LIN {X 0,Y 486.254,Z 781.859,A -85,B 0,C 180,E1 22613.17,E2 22613.17} C_VEL
LIN {X 0,Y 485.416,Z 799.484,A -85,B 0,C 180,E1 22612.272,E2 22612.272} C_VEL
LIN {X 0,Y 484.471,Z 816.535,A -85,B 0,C 180,E1 22611.172,E2 22611.172} C_VEL
LIN {X 0,Y 483.537,Z 833.395,A -85,B 0,C 180,E1 22609.824,E2 22609.824} C_VEL
LIN {X 0,Y 482.628,Z 848.999,A -85,B 0,C 180,E1 22608.302,E2 22608.302} C_VEL
LIN {X 0,Y 481.853,Z 863.116,A -85,B 0,C 180,E1 22606.64,E2 22606.64} C_VEL
LIN {X 0,Y 481.192,Z 876.044,A -85,B 0,C 180,E1 22604.808,E2 22604.808} C_VEL
LIN {X 0,Y 480.699,Z 887.391,A -85,B 0,C 180,E1 22602.86,E2 22602.86} C_VEL
LIN {X 0,Y 480.358,Z 897.146,A -85,B 0,C 180,E1 22600.797,E2 22600.797} C_VEL
LIN {X 0,Y 480.152,Z 905.245,A -85,B 0,C 180,E1 22598.623,E2 22598.623} C_VEL
LIN {X 0,Y 480.072,Z 911.354,A -85,B 0,C 180,E1 22596.458,E2 22596.458} C_VEL
LIN {X 0,Y 480.048,Z 915.622,A -85,B 0,C 180,E1 22594.3,E2 22594.3} C_VEL
LIN {X 0,Y 480.043,Z 918.148,A -85,B 0,C 180,E1 22592.149,E2 22592.149} C_VEL
LIN {X 0,Y 480.045,Z 918.986,A -85,B 0,C 180,E1 22590,E2 22590} C_VEL
LIN {X 0,Y 480.041,Z 918.046,A -85,B 0,C 180,E1 22587.732,E2 22587.732} C_VEL
LIN {X 0,Y 480.048,Z 915.422,A -85,B 0,C 180,E1 22585.58,E2 22585.58} C_VEL
LIN {X 0,Y 480.074,Z 911.042,A -85,B 0,C 180,E1 22583.423,E2 22583.423} C_VEL
LIN {X 0,Y 480.159,Z 904.804,A -85,B 0,C 180,E1 22581.257,E2 22581.257} C_VEL
LIN {X 0,Y 480.363,Z 897.052,A -85,B 0,C 180,E1 22579.203,E2 22579.203} C_VEL
LIN {X 0,Y 480.7,Z 887.258,A -85,B 0,C 180,E1 22577.141,E2 22577.141} C_VEL
LIN {X 0,Y 481.191,Z 875.865,A -85,B 0,C 180,E1 22575.192,E2 22575.192} C_VEL
LIN {X 0,Y 481.823,Z 863.363,A -85,B 0,C 180,E1 22573.421,E2 22573.421} C_VEL
LIN {X 0,Y 482.577,Z 849.357,A -85,B 0,C 180,E1 22571.769,E2 22571.769} C_VEL
LIN {X 0,Y 483.439,Z 834.399,A -85,B 0,C 180,E1 22570.299,E2 22570.299} C_VEL
LIN {X 0,Y 484.304,Z 818.578,A -85,B 0,C 180,E1 22569.011,E2 22569.011} C_VEL
LIN {X 0,Y 485.221,Z 801.998,A -85,B 0,C 180,E1 22567.91,E2 22567.91} C_VEL
LIN {X 0,Y 486.072,Z 783.949,A -85,B 0,C 180,E1 22566.959,E2 22566.959} C_VEL
LIN {X 0,Y 486.851,Z 764.903,A -85,B 0,C 180,E1 22566.207,E2 22566.207} C_VEL
LIN {X 0,Y 487.467,Z 746.066,A -85,B 0,C 180,E1 22565.697,E2 22565.697} C_VEL
LIN {X 0,Y 487.855,Z 712.64,A -85,B 0,C 180,E1 22565.166,E2 22565.166} C_VEL
LIN {X 0,Y 489.112,Z 554.122,A -85,B 0,C 180,E1 22562.794,E2 22562.794} C_VEL
LIN {X 0,Y 487.309,Z 539.68,A -85,B 0,C 180,E1 22562.457,E2 22562.457} C_VEL
LIN {X 0,Y 489.579,Z 496.19,A -85,B 0,C 180,E1 22558.839,E2 22558.839} C_VEL
LIN {X 0,Y 490.971,Z 471.845,A -85,B 0,C 180,E1 22556.729,E2 22556.729} C_VEL
LIN {X 0,Y 484.233,Z 452.154,A -85,B 0,C 180,E1 22554.342,E2 22554.342} C_VEL
LIN {X 0,Y 480.918,Z 443.105,A -85,B 0,C 180,E1 22553.11,E2 22553.11} C_VEL
LIN {X 0,Y 480.88,Z 442.893,A -85,B 0,C 180,E1 22549.552,E2 22549.552} C_VEL
LIN {X 0,Y 480.889,Z 442.899,A -85,B 0,C 180,E1 22546.005,E2 22546.005} C_VEL
LIN {X 0,Y 480.884,Z 442.893,A -85,B 0,C 180,E1 22542.35,E2 22542.35} C_VEL
LIN {X 0,Y 480.891,Z 442.887,A -85,B 0,C 180,E1 22538.743,E2 22538.743} C_VEL
LIN {X 0,Y 480.877,Z 442.894,A -85,B 0,C 180,E1 22535.166,E2 22535.166} C_VEL
LIN {X 0,Y 480.881,Z 442.893,A -85,B 0,C 180,E1 22531.518,E2 22531.518} C_VEL
LIN {X 0,Y 480.889,Z 442.887,A -85,B 0,C 180,E1 22527.893,E2 22527.893} C_VEL
LIN {X 0,Y 480.886,Z 442.888,A -85,B 0,C 180,E1 22524.31,E2 22524.31} C_VEL
LIN {X 0,Y 480.883,Z 442.891,A -85,B 0,C 180,E1 22520.699,E2 22520.699} C_VEL
LIN {X 0,Y 480.876,Z 442.897,A -85,B 0,C 180,E1 22517.048,E2 22517.048} C_VEL
LIN {X 0,Y 480.889,Z 442.888,A -85,B 0,C 180,E1 22513.466,E2 22513.466} C_VEL
LIN {X 0,Y 480.884,Z 442.886,A -85,B 0,C 180,E1 22509.816,E2 22509.816} C_VEL
LIN {X 0,Y 480.888,Z 442.891,A -85,B 0,C 180,E1 22506.207,E2 22506.207} C_VEL
LIN {X 0,Y 480.873,Z 442.896,A -85,B 0,C 180,E1 22502.622,E2 22502.622} C_VEL
LIN {X 0,Y 480.887,Z 442.888,A -85,B 0,C 180,E1 22499.047,E2 22499.047} C_VEL
LIN {X 0,Y 480.885,Z 442.889,A -85,B 0,C 180,E1 22495.468,E2 22495.468} C_VEL
LIN {X 0,Y 480.889,Z 442.892,A -85,B 0,C 180,E1 22491.872,E2 22491.872} C_VEL
LIN {X 0,Y 480.872,Z 442.896,A -85,B 0,C 180,E1 22488.242,E2 22488.242} C_VEL
LIN {X 0,Y 480.879,Z 442.899,A -85,B 0,C 180,E1 22484.565,E2 22484.565} C_VEL
LIN {X 0,Y 480.888,Z 442.895,A -85,B 0,C 180,E1 22480.947,E2 22480.947} C_VEL
LIN {X 0,Y 480.893,Z 442.894,A -85,B 0,C 180,E1 22477.378,E2 22477.378} C_VEL
LIN {X 0,Y 480.873,Z 442.897,A -85,B 0,C 180,E1 22473.845,E2 22473.845} C_VEL
LIN {X 0,Y 480.876,Z 442.894,A -85,B 0,C 180,E1 22470.202,E2 22470.202} C_VEL
LIN {X 0,Y 480.892,Z 442.899,A -85,B 0,C 180,E1 22466.565,E2 22466.565} C_VEL
LIN {X 0,Y 480.89,Z 442.9,A -85,B 0,C 180,E1 22462.917,E2 22462.917} C_VEL
LIN {X 0,Y 480.983,Z 443.47,A -85,B 0,C 180,E1 22462.626,E2 22462.626} C_VEL
LIN {X 0,Y 485.678,Z 459.122,A -85,B 0,C 180,E1 22459.981,E2 22459.981} C_VEL
LIN {X 0,Y 487.767,Z 467.746,A -85,B 0,C 180,E1 22458.612,E2 22458.612} C_VEL
LIN {X 0,Y 485.992,Z 496.046,A -85,B 0,C 180,E1 22454.884,E2 22454.884} C_VEL
LIN {X 0,Y 484.498,Z 525.084,A -85,B 0,C 180,E1 22451.127,E2 22451.127} C_VEL
LIN {X 0,Y 483.217,Z 552.995,A -85,B 0,C 180,E1 22447.58,E2 22447.58} C_VEL
LIN {X 0,Y 483.229,Z 556.14,A -85,B 0,C 180,E1 22447.246,E2 22447.246} C_VEL
LIN {X 0,Y 484.694,Z 563.985,A -85,B 0,C 180,E1 22447.03,E2 22447.03} C_VEL
LIN {X 0,Y 484.537,Z 568.371,A -85,B 0,C 180,E1 22446.968,E2 22446.968} C_VEL
LIN {X 0,Y 481.971,Z 575.469,A -85,B 0,C 180,E1 22446.983,E2 22446.983} C_VEL
LIN {X 0,Y 478.786,Z 583.343,A -85,B 0,C 180,E1 22447.017,E2 22447.017} C_VEL
LIN {X 0,Y 478.245,Z 587.099,A -85,B 0,C 180,E1 22446.983,E2 22446.983} C_VEL
LIN {X 0,Y 477.175,Z 673.778,A -85,B 0,C 180,E1 22445.564,E2 22445.564} C_VEL
LIN {X 0,Y 476.885,Z 688.496,A -85,B 0,C 180,E1 22445.107,E2 22445.107} C_VEL
LIN {X 0,Y 476.416,Z 702.899,A -85,B 0,C 180,E1 22444.432,E2 22444.432} C_VEL
LIN {X 0,Y 475.812,Z 716.66,A -85,B 0,C 180,E1 22443.55,E2 22443.55} C_VEL
LIN {X 0,Y 475.116,Z 729.674,A -85,B 0,C 180,E1 22442.447,E2 22442.447} C_VEL
LIN {X 0,Y 474.5,Z 740.893,A -85,B 0,C 180,E1 22441.223,E2 22441.223} C_VEL
LIN {X 0,Y 473.923,Z 750.816,A -85,B 0,C 180,E1 22439.861,E2 22439.861} C_VEL
LIN {X 0,Y 473.385,Z 759.978,A -85,B 0,C 180,E1 22438.237,E2 22438.237} C_VEL
LIN {X 0,Y 472.992,Z 767.015,A -85,B 0,C 180,E1 22436.596,E2 22436.596} C_VEL
LIN {X 0,Y 472.72,Z 772.499,A -85,B 0,C 180,E1 22434.853,E2 22434.853} C_VEL
LIN {X 0,Y 472.548,Z 776.275,A -85,B 0,C 180,E1 22433.013,E2 22433.013} C_VEL
LIN {X 0,Y 472.471,Z 778.221,A -85,B 0,C 180,E1 22431.215,E2 22431.215} C_VEL
LIN {X 0,Y 472.455,Z 778.461,A -85,B 0,C 180,E1 22429.277,E2 22429.277} C_VEL
LIN {X 0,Y 472.497,Z 776.776,A -85,B 0,C 180,E1 22427.36,E2 22427.36} C_VEL
LIN {X 0,Y 472.617,Z 773.493,A -85,B 0,C 180,E1 22425.585,E2 22425.585} C_VEL
LIN {X 0,Y 472.837,Z 768.431,A -85,B 0,C 180,E1 22423.824,E2 22423.824} C_VEL
LIN {X 0,Y 473.157,Z 761.926,A -85,B 0,C 180,E1 22422.199,E2 22422.199} C_VEL
LIN {X 0,Y 473.614,Z 753.426,A -85,B 0,C 180,E1 22420.583,E2 22420.583} C_VEL
LIN {X 0,Y 474.176,Z 743.294,A -85,B 0,C 180,E1 22419.099,E2 22419.099} C_VEL
LIN {X 0,Y 474.788,Z 731.95,A -85,B 0,C 180,E1 22417.801,E2 22417.801} C_VEL
LIN {X 0,Y 475.406,Z 719.74,A -85,B 0,C 180,E1 22416.703,E2 22416.703} C_VEL
LIN {X 0,Y 476.041,Z 705.469,A -85,B 0,C 180,E1 22415.726,E2 22415.726} C_VEL
LIN {X 0,Y 476.539,Z 690.725,A -85,B 0,C 180,E1 22414.995,E2 22414.995} C_VEL
LIN {X 0,Y 476.872,Z 676.023,A -85,B 0,C 180,E1 22414.502,E2 22414.502} C_VEL
LIN {X 0,Y 477.117,Z 653.857,A -85,B 0,C 180,E1 22414.095,E2 22414.095} C_VEL
LIN {X 0,Y 477.797,Z 569.714,A -85,B 0,C 180,E1 22412.77,E2 22412.77} C_VEL
LIN {X 0,Y 475.295,Z 555.743,A -85,B 0,C 180,E1 22412.411,E2 22412.411} C_VEL
LIN {X 0,Y 476.452,Z 528.148,A -85,B 0,C 180,E1 22408.918,E2 22408.918} C_VEL
LIN {X 0,Y 477.91,Z 500.312,A -85,B 0,C 180,E1 22405.32,E2 22405.32} C_VEL
LIN {X 0,Y 479.613,Z 471.177,A -85,B 0,C 180,E1 22401.488,E2 22401.488} C_VEL
LIN {X 0,Y 479.507,Z 467.664,A -85,B 0,C 180,E1 22401.002,E2 22401.002} C_VEL
LIN {X 0,Y 474.285,Z 448.82,A -85,B 0,C 180,E1 22398.01,E2 22398.01} C_VEL
LIN {X 0,Y 472.919,Z 444,A -85,B 0,C 180,E1 22397.174,E2 22397.174} C_VEL
LIN {X 0,Y 472.938,Z 443.888,A -85,B 0,C 180,E1 22393.669,E2 22393.669} C_VEL
LIN {X 0,Y 472.892,Z 443.888,A -85,B 0,C 180,E1 22390.098,E2 22390.098} C_VEL
LIN {X 0,Y 472.875,Z 443.865,A -85,B 0,C 180,E1 22386.577,E2 22386.577} C_VEL
LIN {X 0,Y 472.911,Z 443.889,A -85,B 0,C 180,E1 22383.099,E2 22383.099} C_VEL
LIN {X 0,Y 472.909,Z 443.891,A -85,B 0,C 180,E1 22379.613,E2 22379.613} C_VEL
LIN {X 0,Y 472.871,Z 443.89,A -85,B 0,C 180,E1 22376.2,E2 22376.2} C_VEL
LIN {X 0,Y 472.889,Z 443.885,A -85,B 0,C 180,E1 22372.64,E2 22372.64} C_VEL
LIN {X 0,Y 472.942,Z 443.882,A -85,B 0,C 180,E1 22369.188,E2 22369.188} C_VEL
LIN {X 0,Y 472.898,Z 443.887,A -85,B 0,C 180,E1 22365.585,E2 22365.585} C_VEL
LIN {X 0,Y 472.882,Z 443.878,A -85,B 0,C 180,E1 22362.085,E2 22362.085} C_VEL
LIN {X 0,Y 472.916,Z 443.888,A -85,B 0,C 180,E1 22358.587,E2 22358.587} C_VEL
LIN {X 0,Y 472.928,Z 443.873,A -85,B 0,C 180,E1 22355.095,E2 22355.095} C_VEL
LIN {X 0,Y 472.894,Z 443.886,A -85,B 0,C 180,E1 22351.561,E2 22351.561} C_VEL
LIN {X 0,Y 472.893,Z 443.88,A -85,B 0,C 180,E1 22347.896,E2 22347.896} C_VEL
LIN {X 0,Y 472.927,Z 443.882,A -85,B 0,C 180,E1 22344.348,E2 22344.348} C_VEL
LIN {X 0,Y 472.944,Z 443.885,A -85,B 0,C 180,E1 22340.804,E2 22340.804} C_VEL
LIN {X 0,Y 472.905,Z 443.865,A -85,B 0,C 180,E1 22337.218,E2 22337.218} C_VEL
LIN {X 0,Y 472.903,Z 443.886,A -85,B 0,C 180,E1 22333.573,E2 22333.573} C_VEL
LIN {X 0,Y 472.926,Z 443.869,A -85,B 0,C 180,E1 22329.984,E2 22329.984} C_VEL
LIN {X 0,Y 472.956,Z 443.877,A -85,B 0,C 180,E1 22326.433,E2 22326.433} C_VEL
LIN {X 0,Y 472.927,Z 443.887,A -85,B 0,C 180,E1 22322.787,E2 22322.787} C_VEL
LIN {X 0,Y 472.908,Z 443.87,A -85,B 0,C 180,E1 22319.273,E2 22319.273} C_VEL
LIN {X 0,Y 472.937,Z 443.883,A -85,B 0,C 180,E1 22315.757,E2 22315.757} C_VEL
LIN {X 0,Y 472.954,Z 443.867,A -85,B 0,C 180,E1 22312.102,E2 22312.102} C_VEL
LIN {X 0,Y 472.942,Z 443.888,A -85,B 0,C 180,E1 22308.414,E2 22308.414} C_VEL
LIN {X 0,Y 472.919,Z 443.872,A -85,B 0,C 180,E1 22304.802,E2 22304.802} C_VEL
LIN {X 0,Y 472.926,Z 443.884,A -85,B 0,C 180,E1 22301.127,E2 22301.127} C_VEL
LIN {X 0,Y 472.954,Z 443.877,A -85,B 0,C 180,E1 22297.496,E2 22297.496} C_VEL
LIN {X 0,Y 472.951,Z 443.874,A -85,B 0,C 180,E1 22293.779,E2 22293.779} C_VEL
LIN {X 0,Y 472.952,Z 443.887,A -85,B 0,C 180,E1 22290.071,E2 22290.071} C_VEL
LIN {X 0,Y 472.933,Z 443.885,A -85,B 0,C 180,E1 22286.407,E2 22286.407} C_VEL
LIN {X 0,Y 472.934,Z 443.884,A -85,B 0,C 180,E1 22282.796,E2 22282.796} C_VEL
LIN {X 0,Y 472.958,Z 443.883,A -85,B 0,C 180,E1 22279.186,E2 22279.186} C_VEL
LIN {X 0,Y 472.948,Z 443.882,A -85,B 0,C 180,E1 22275.435,E2 22275.435} C_VEL
LIN {X 0,Y 472.951,Z 443.884,A -85,B 0,C 180,E1 22271.732,E2 22271.732} C_VEL
LIN {X 0,Y 472.939,Z 443.883,A -85,B 0,C 180,E1 22268.122,E2 22268.122} C_VEL
LIN {X 0,Y 472.985,Z 444.157,A -85,B 0,C 180,E1 22267.16,E2 22267.16} C_VEL
LIN {X 0,Y 481.537,Z 468.501,A -85,B 0,C 180,E1 22264.163,E2 22264.163} C_VEL
LIN {X 0,Y 483.625,Z 474.838,A -85,B 0,C 180,E1 22263.434,E2 22263.434} C_VEL
LIN {X 0,Y 480.864,Z 519.742,A -85,B 0,C 180,E1 22259.593,E2 22259.593} C_VEL
LIN {X 0,Y 479.862,Z 540.27,A -85,B 0,C 180,E1 22257.9,E2 22257.9} C_VEL
LIN {X 0,Y 481.929,Z 558.241,A -85,B 0,C 180,E1 22257.511,E2 22257.511} C_VEL
LIN {X 0,Y 480.036,Z 744.193,A -85,B 0,C 180,E1 22254.685,E2 22254.685} C_VEL
LIN {X 0,Y 479.411,Z 763.112,A -85,B 0,C 180,E1 22254.181,E2 22254.181} C_VEL
LIN {X 0,Y 478.653,Z 780.656,A -85,B 0,C 180,E1 22253.505,E2 22253.505} C_VEL
LIN {X 0,Y 477.74,Z 798.568,A -85,B 0,C 180,E1 22252.585,E2 22252.585} C_VEL
LIN {X 0,Y 476.738,Z 815.637,A -85,B 0,C 180,E1 22251.468,E2 22251.468} C_VEL
LIN {X 0,Y 475.781,Z 831.799,A -85,B 0,C 180,E1 22250.161,E2 22250.161} C_VEL
LIN {X 0,Y 474.811,Z 847.377,A -85,B 0,C 180,E1 22248.628,E2 22248.628} C_VEL
LIN {X 0,Y 473.965,Z 861.701,A -85,B 0,C 180,E1 22246.925,E2 22246.925} C_VEL
LIN {X 0,Y 473.275,Z 874.449,A -85,B 0,C 180,E1 22245.1,E2 22245.1} C_VEL
LIN {X 0,Y 472.774,Z 885.424,A -85,B 0,C 180,E1 22243.204,E2 22243.204} C_VEL
LIN {X 0,Y 472.433,Z 894.819,A -85,B 0,C 180,E1 22241.228,E2 22241.228} C_VEL
LIN {X 0,Y 472.215,Z 902.799,A -85,B 0,C 180,E1 22239.138,E2 22239.138} C_VEL
LIN {X 0,Y 472.129,Z 908.944,A -85,B 0,C 180,E1 22237.056,E2 22237.056} C_VEL
LIN {X 0,Y 472.109,Z 913.627,A -85,B 0,C 180,E1 22234.86,E2 22234.86} C_VEL
LIN {X 0,Y 472.115,Z 916.533,A -85,B 0,C 180,E1 22232.671,E2 22232.671} C_VEL
LIN {X 0,Y 472.125,Z 917.735,A -85,B 0,C 180,E1 22230.486,E2 22230.486} C_VEL
LIN {X 0,Y 472.127,Z 917.257,A -85,B 0,C 180,E1 22228.301,E2 22228.301} C_VEL
LIN {X 0,Y 472.122,Z 915.092,A -85,B 0,C 180,E1 22226.114,E2 22226.114} C_VEL
LIN {X 0,Y 472.126,Z 911.188,A -85,B 0,C 180,E1 22223.922,E2 22223.922} C_VEL
LIN {X 0,Y 472.181,Z 905.446,A -85,B 0,C 180,E1 22221.721,E2 22221.721} C_VEL
LIN {X 0,Y 472.347,Z 897.72,A -85,B 0,C 180,E1 22219.511,E2 22219.511} C_VEL
LIN {X 0,Y 472.65,Z 888.391,A -85,B 0,C 180,E1 22217.415,E2 22217.415} C_VEL
LIN {X 0,Y 473.11,Z 877.522,A -85,B 0,C 180,E1 22215.434,E2 22215.434} C_VEL
LIN {X 0,Y 473.755,Z 865.138,A -85,B 0,C 180,E1 22213.572,E2 22213.572} C_VEL
LIN {X 0,Y 474.547,Z 851.184,A -85,B 0,C 180,E1 22211.831,E2 22211.831} C_VEL
LIN {X 0,Y 475.471,Z 836.163,A -85,B 0,C 180,E1 22210.275,E2 22210.275} C_VEL
LIN {X 0,Y 476.415,Z 820.117,A -85,B 0,C 180,E1 22208.904,E2 22208.904} C_VEL
LIN {X 0,Y 477.425,Z 803.102,A -85,B 0,C 180,E1 22207.725,E2 22207.725} C_VEL
LIN {X 0,Y 478.321,Z 785.678,A -85,B 0,C 180,E1 22206.762,E2 22206.762} C_VEL
LIN {X 0,Y 479.158,Z 767.387,A -85,B 0,C 180,E1 22205.994,E2 22205.994} C_VEL
LIN {X 0,Y 479.849,Z 748.623,A -85,B 0,C 180,E1 22205.441,E2 22205.441} C_VEL
LIN {X 0,Y 480.227,Z 725.573,A -85,B 0,C 180,E1 22205.031,E2 22205.031} C_VEL
LIN {X 0,Y 481.699,Z 555.105,A -85,B 0,C 180,E1 22202.447,E2 22202.447} C_VEL
LIN {X 0,Y 479.837,Z 539.958,A -85,B 0,C 180,E1 22202.09,E2 22202.09} C_VEL
LIN {X 0,Y 482.352,Z 496.151,A -85,B 0,C 180,E1 22198.37,E2 22198.37} C_VEL
LIN {X 0,Y 483.845,Z 475.048,A -85,B 0,C 180,E1 22196.513,E2 22196.513} C_VEL
LIN {X 0,Y 477.379,Z 456.001,A -85,B 0,C 180,E1 22194.151,E2 22194.151} C_VEL
LIN {X 0,Y 472.978,Z 444.121,A -85,B 0,C 180,E1 22192.496,E2 22192.496} C_VEL
LIN {X 0,Y 472.955,Z 443.881,A -85,B 0,C 180,E1 22189.001,E2 22189.001} C_VEL
LIN {X 0,Y 472.941,Z 443.882,A -85,B 0,C 180,E1 22185.421,E2 22185.421} C_VEL
LIN {X 0,Y 472.943,Z 443.882,A -85,B 0,C 180,E1 22181.731,E2 22181.731} C_VEL
LIN {X 0,Y 472.948,Z 443.882,A -85,B 0,C 180,E1 22178.12,E2 22178.12} C_VEL
LIN {X 0,Y 472.947,Z 443.883,A -85,B 0,C 180,E1 22174.462,E2 22174.462} C_VEL
LIN {X 0,Y 472.952,Z 443.881,A -85,B 0,C 180,E1 22170.771,E2 22170.771} C_VEL
LIN {X 0,Y 472.938,Z 443.884,A -85,B 0,C 180,E1 22167.12,E2 22167.12} C_VEL
LIN {X 0,Y 472.944,Z 443.877,A -85,B 0,C 180,E1 22163.419,E2 22163.419} C_VEL
LIN {X 0,Y 472.947,Z 443.876,A -85,B 0,C 180,E1 22159.771,E2 22159.771} C_VEL
LIN {X 0,Y 472.95,Z 443.883,A -85,B 0,C 180,E1 22156.078,E2 22156.078} C_VEL
LIN {X 0,Y 472.948,Z 443.882,A -85,B 0,C 180,E1 22152.39,E2 22152.39} C_VEL
LIN {X 0,Y 472.934,Z 443.881,A -85,B 0,C 180,E1 22148.755,E2 22148.755} C_VEL
LIN {X 0,Y 472.944,Z 443.873,A -85,B 0,C 180,E1 22145.094,E2 22145.094} C_VEL
LIN {X 0,Y 472.949,Z 443.887,A -85,B 0,C 180,E1 22141.453,E2 22141.453} C_VEL
LIN {X 0,Y 472.949,Z 443.881,A -85,B 0,C 180,E1 22137.819,E2 22137.819} C_VEL
LIN {X 0,Y 472.938,Z 443.878,A -85,B 0,C 180,E1 22134.175,E2 22134.175} C_VEL
LIN {X 0,Y 472.933,Z 443.875,A -85,B 0,C 180,E1 22130.508,E2 22130.508} C_VEL
LIN {X 0,Y 472.951,Z 443.878,A -85,B 0,C 180,E1 22126.926,E2 22126.926} C_VEL
LIN {X 0,Y 472.95,Z 443.885,A -85,B 0,C 180,E1 22123.272,E2 22123.272} C_VEL
LIN {X 0,Y 472.95,Z 443.881,A -85,B 0,C 180,E1 22119.584,E2 22119.584} C_VEL
LIN {X 0,Y 472.932,Z 443.879,A -85,B 0,C 180,E1 22115.968,E2 22115.968} C_VEL
LIN {X 0,Y 472.938,Z 443.883,A -85,B 0,C 180,E1 22112.282,E2 22112.282} C_VEL
LIN {X 0,Y 472.953,Z 443.888,A -85,B 0,C 180,E1 22108.659,E2 22108.659} C_VEL
LIN {X 0,Y 472.95,Z 443.885,A -85,B 0,C 180,E1 22105.046,E2 22105.046} C_VEL
LIN {X 0,Y 472.987,Z 444.168,A -85,B 0,C 180,E1 22103.265,E2 22103.265} C_VEL
LIN {X 0,Y 477.786,Z 460.078,A -85,B 0,C 180,E1 22100.492,E2 22100.492} C_VEL
LIN {X 0,Y 480.357,Z 470.628,A -85,B 0,C 180,E1 22098.784,E2 22098.784} C_VEL
LIN {X 0,Y 478.473,Z 498.449,A -85,B 0,C 180,E1 22095.064,E2 22095.064} C_VEL
LIN {X 0,Y 476.851,Z 527.78,A -85,B 0,C 180,E1 22091.219,E2 22091.219} C_VEL
LIN {X 0,Y 475.541,Z 555.513,A -85,B 0,C 180,E1 22087.672,E2 22087.672} C_VEL
LIN {X 0,Y 478.414,Z 572.463,A -85,B 0,C 180,E1 22087.211,E2 22087.211} C_VEL
LIN {X 0,Y 478.245,Z 587.099,A -85,B 0,C 180,E1 22086.983,E2 22086.983} C_VEL
LIN {X 0,Y 477.253,Z 594.774,A -85,B 0,C 180,E1 22086.908,E2 22086.908} C_VEL
LIN {X 0,Y 471.199,Z 615.147,A -85,B 0,C 180,E1 22086.879,E2 22086.879} C_VEL
LIN {X 0,Y 470.418,Z 621.736,A -85,B 0,C 180,E1 22086.808,E2 22086.808} C_VEL
LIN {X 0,Y 469.706,Z 674.934,A -85,B 0,C 180,E1 22085.892,E2 22085.892} C_VEL
LIN {X 0,Y 469.383,Z 689.984,A -85,B 0,C 180,E1 22085.408,E2 22085.408} C_VEL
LIN {X 0,Y 468.844,Z 704.953,A -85,B 0,C 180,E1 22084.677,E2 22084.677} C_VEL
LIN {X 0,Y 468.21,Z 718.149,A -85,B 0,C 180,E1 22083.8,E2 22083.8} C_VEL
LIN {X 0,Y 467.466,Z 731.164,A -85,B 0,C 180,E1 22082.67,E2 22082.67} C_VEL
LIN {X 0,Y 466.768,Z 742.733,A -85,B 0,C 180,E1 22081.367,E2 22081.367} C_VEL
LIN {X 0,Y 466.124,Z 752.784,A -85,B 0,C 180,E1 22079.933,E2 22079.933} C_VEL
LIN {X 0,Y 465.557,Z 761.73,A -85,B 0,C 180,E1 22078.292,E2 22078.292} C_VEL
LIN {X 0,Y 465.114,Z 768.817,A -85,B 0,C 180,E1 22076.56,E2 22076.56} C_VEL
LIN {X 0,Y 464.823,Z 774.054,A -85,B 0,C 180,E1 22074.8,E2 22074.8} C_VEL
LIN {X 0,Y 464.643,Z 777.701,A -85,B 0,C 180,E1 22072.923,E2 22072.923} C_VEL
LIN {X 0,Y 464.556,Z 779.486,A -85,B 0,C 180,E1 22071.065,E2 22071.065} C_VEL
LIN {X 0,Y 464.542,Z 779.612,A -85,B 0,C 180,E1 22069.227,E2 22069.227} C_VEL
LIN {X 0,Y 464.591,Z 777.883,A -85,B 0,C 180,E1 22067.277,E2 22067.277} C_VEL
LIN {X 0,Y 464.727,Z 774.5,A -85,B 0,C 180,E1 22065.447,E2 22065.447} C_VEL
LIN {X 0,Y 464.989,Z 769.223,A -85,B 0,C 180,E1 22063.606,E2 22063.606} C_VEL
LIN {X 0,Y 465.362,Z 762.364,A -85,B 0,C 180,E1 22061.903,E2 22061.903} C_VEL
LIN {X 0,Y 465.828,Z 754.423,A -85,B 0,C 180,E1 22060.387,E2 22060.387} C_VEL
LIN {X 0,Y 466.464,Z 743.904,A -85,B 0,C 180,E1 22058.828,E2 22058.828} C_VEL
LIN {X 0,Y 467.13,Z 732.376,A -85,B 0,C 180,E1 22057.502,E2 22057.502} C_VEL
LIN {X 0,Y 467.763,Z 720.743,A -85,B 0,C 180,E1 22056.443,E2 22056.443} C_VEL
LIN {X 0,Y 468.438,Z 706.507,A -85,B 0,C 180,E1 22055.45,E2 22055.45} C_VEL
LIN {X 0,Y 468.944,Z 692.617,A -85,B 0,C 180,E1 22054.739,E2 22054.739} C_VEL
LIN {X 0,Y 469.327,Z 677.402,A -85,B 0,C 180,E1 22054.203,E2 22054.203} C_VEL
LIN {X 0,Y 469.58,Z 656.344,A -85,B 0,C 180,E1 22053.8,E2 22053.8} C_VEL
LIN {X 0,Y 470.338,Z 570.745,A -85,B 0,C 180,E1 22052.427,E2 22052.427} C_VEL
LIN {X 0,Y 467.618,Z 555.442,A -85,B 0,C 180,E1 22052.022,E2 22052.022} C_VEL
LIN {X 0,Y 468.986,Z 525.511,A -85,B 0,C 180,E1 22048.167,E2 22048.167} C_VEL
LIN {X 0,Y 470.632,Z 496.716,A -85,B 0,C 180,E1 22044.391,E2 22044.391} C_VEL
LIN {X 0,Y 472.237,Z 471.169,A -85,B 0,C 180,E1 22040.986,E2 22040.986} C_VEL
LIN {X 0,Y 467.419,Z 453.515,A -85,B 0,C 180,E1 22038.15,E2 22038.15} C_VEL
LIN {X 0,Y 464.961,Z 445.004,A -85,B 0,C 180,E1 22036.697,E2 22036.697} C_VEL
LIN {X 0,Y 464.975,Z 444.875,A -85,B 0,C 180,E1 22033.253,E2 22033.253} C_VEL
LIN {X 0,Y 464.994,Z 444.877,A -85,B 0,C 180,E1 22029.614,E2 22029.614} C_VEL
LIN {X 0,Y 464.94,Z 444.854,A -85,B 0,C 180,E1 22026.153,E2 22026.153} C_VEL
LIN {X 0,Y 464.938,Z 444.877,A -85,B 0,C 180,E1 22022.599,E2 22022.599} C_VEL
LIN {X 0,Y 464.976,Z 444.875,A -85,B 0,C 180,E1 22019.092,E2 22019.092} C_VEL
LIN {X 0,Y 464.979,Z 444.88,A -85,B 0,C 180,E1 22015.445,E2 22015.445} C_VEL
LIN {X 0,Y 464.942,Z 444.875,A -85,B 0,C 180,E1 22011.888,E2 22011.888} C_VEL
LIN {X 0,Y 464.939,Z 444.869,A -85,B 0,C 180,E1 22008.265,E2 22008.265} C_VEL
LIN {X 0,Y 464.982,Z 444.878,A -85,B 0,C 180,E1 22004.797,E2 22004.797} C_VEL
LIN {X 0,Y 464.994,Z 444.861,A -85,B 0,C 180,E1 22001.146,E2 22001.146} C_VEL
LIN {X 0,Y 464.953,Z 444.879,A -85,B 0,C 180,E1 21997.643,E2 21997.643} C_VEL
LIN {X 0,Y 464.949,Z 444.859,A -85,B 0,C 180,E1 21993.996,E2 21993.996} C_VEL
LIN {X 0,Y 464.982,Z 444.876,A -85,B 0,C 180,E1 21990.426,E2 21990.426} C_VEL
LIN {X 0,Y 465.004,Z 444.854,A -85,B 0,C 180,E1 21986.843,E2 21986.843} C_VEL
LIN {X 0,Y 464.966,Z 444.873,A -85,B 0,C 180,E1 21983.308,E2 21983.308} C_VEL
LIN {X 0,Y 464.96,Z 444.869,A -85,B 0,C 180,E1 21979.732,E2 21979.732} C_VEL
LIN {X 0,Y 464.985,Z 444.865,A -85,B 0,C 180,E1 21976.105,E2 21976.105} C_VEL
LIN {X 0,Y 465.013,Z 444.873,A -85,B 0,C 180,E1 21972.53,E2 21972.53} C_VEL
LIN {X 0,Y 464.981,Z 444.854,A -85,B 0,C 180,E1 21968.907,E2 21968.907} C_VEL
LIN {X 0,Y 464.969,Z 444.873,A -85,B 0,C 180,E1 21965.306,E2 21965.306} C_VEL
LIN {X 0,Y 464.983,Z 444.861,A -85,B 0,C 180,E1 21961.725,E2 21961.725} C_VEL
LIN {X 0,Y 465.014,Z 444.867,A -85,B 0,C 180,E1 21958.152,E2 21958.152} C_VEL
LIN {X 0,Y 465.004,Z 444.871,A -85,B 0,C 180,E1 21954.448,E2 21954.448} C_VEL
LIN {X 0,Y 464.98,Z 444.862,A -85,B 0,C 180,E1 21950.844,E2 21950.844} C_VEL
LIN {X 0,Y 464.982,Z 444.872,A -85,B 0,C 180,E1 21947.204,E2 21947.204} C_VEL
LIN {X 0,Y 465.01,Z 444.867,A -85,B 0,C 180,E1 21943.64,E2 21943.64} C_VEL
LIN {X 0,Y 465.014,Z 444.866,A -85,B 0,C 180,E1 21939.989,E2 21939.989} C_VEL
LIN {X 0,Y 464.999,Z 444.873,A -85,B 0,C 180,E1 21936.349,E2 21936.349} C_VEL
LIN {X 0,Y 464.985,Z 444.862,A -85,B 0,C 180,E1 21932.741,E2 21932.741} C_VEL
LIN {X 0,Y 465,Z 444.868,A -85,B 0,C 180,E1 21929.076,E2 21929.076} C_VEL
LIN {X 0,Y 465.011,Z 444.87,A -85,B 0,C 180,E1 21925.414,E2 21925.414} C_VEL
LIN {X 0,Y 465.013,Z 444.871,A -85,B 0,C 180,E1 21921.704,E2 21921.704} C_VEL
LIN {X 0,Y 465.006,Z 444.872,A -85,B 0,C 180,E1 21918.032,E2 21918.032} C_VEL
LIN {X 0,Y 464.996,Z 444.871,A -85,B 0,C 180,E1 21914.334,E2 21914.334} C_VEL
LIN {X 0,Y 465.004,Z 444.875,A -85,B 0,C 180,E1 21910.622,E2 21910.622} C_VEL
LIN {X 0,Y 465.05,Z 445.132,A -85,B 0,C 180,E1 21907.702,E2 21907.702} C_VEL
LIN {X 0,Y 473.284,Z 468.583,A -85,B 0,C 180,E1 21904.735,E2 21904.735} C_VEL
LIN {X 0,Y 476.234,Z 477.742,A -85,B 0,C 180,E1 21903.661,E2 21903.661} C_VEL
LIN {X 0,Y 473.349,Z 521.729,A -85,B 0,C 180,E1 21899.84,E2 21899.84} C_VEL
LIN {X 0,Y 472.382,Z 540.503,A -85,B 0,C 180,E1 21898.271,E2 21898.271} C_VEL
LIN {X 0,Y 474.513,Z 559.142,A -85,B 0,C 180,E1 21897.861,E2 21897.861} C_VEL
LIN {X 0,Y 472.499,Z 743.507,A -85,B 0,C 180,E1 21895.017,E2 21895.017} C_VEL
LIN {X 0,Y 471.846,Z 762.366,A -85,B 0,C 180,E1 21894.509,E2 21894.509} C_VEL
LIN {X 0,Y 470.991,Z 780.676,A -85,B 0,C 180,E1 21893.788,E2 21893.788} C_VEL
LIN {X 0,Y 470.076,Z 797.524,A -85,B 0,C 180,E1 21892.908,E2 21892.908} C_VEL
LIN {X 0,Y 469.019,Z 814.657,A -85,B 0,C 180,E1 21891.774,E2 21891.774} C_VEL
LIN {X 0,Y 467.995,Z 830.863,A -85,B 0,C 180,E1 21890.446,E2 21890.446} C_VEL
LIN {X 0,Y 466.952,Z 846.679,A -85,B 0,C 180,E1 21888.865,E2 21888.865} C_VEL
LIN {X 0,Y 466.091,Z 860.29,A -85,B 0,C 180,E1 21887.22,E2 21887.22} C_VEL
LIN {X 0,Y 465.387,Z 872.537,A -85,B 0,C 180,E1 21885.451,E2 21885.451} C_VEL
LIN {X 0,Y 464.841,Z 883.598,A -85,B 0,C 180,E1 21883.533,E2 21883.533} C_VEL
LIN {X 0,Y 464.486,Z 893.017,A -85,B 0,C 180,E1 21881.548,E2 21881.548} C_VEL
LIN {X 0,Y 464.266,Z 901.146,A -85,B 0,C 180,E1 21879.421,E2 21879.421} C_VEL
LIN {X 0,Y 464.178,Z 907.745,A -85,B 0,C 180,E1 21877.177,E2 21877.177} C_VEL
LIN {X 0,Y 464.173,Z 912.447,A -85,B 0,C 180,E1 21874.943,E2 21874.943} C_VEL
LIN {X 0,Y 464.193,Z 915.365,A -85,B 0,C 180,E1 21872.716,E2 21872.716} C_VEL
LIN {X 0,Y 464.21,Z 916.569,A -85,B 0,C 180,E1 21870.494,E2 21870.494} C_VEL
LIN {X 0,Y 464.21,Z 916.085,A -85,B 0,C 180,E1 21868.272,E2 21868.272} C_VEL
LIN {X 0,Y 464.195,Z 913.905,A -85,B 0,C 180,E1 21866.048,E2 21866.048} C_VEL
LIN {X 0,Y 464.186,Z 909.978,A -85,B 0,C 180,E1 21863.817,E2 21863.817} C_VEL
LIN {X 0,Y 464.226,Z 904.205,A -85,B 0,C 180,E1 21861.578,E2 21861.578} C_VEL
LIN {X 0,Y 464.385,Z 896.441,A -85,B 0,C 180,E1 21859.329,E2 21859.329} C_VEL
LIN {X 0,Y 464.696,Z 887.066,A -85,B 0,C 180,E1 21857.196,E2 21857.196} C_VEL
LIN {X 0,Y 465.183,Z 876.143,A -85,B 0,C 180,E1 21855.181,E2 21855.181} C_VEL
LIN {X 0,Y 465.865,Z 863.694,A -85,B 0,C 180,E1 21853.286,E2 21853.286} C_VEL
LIN {X 0,Y 466.71,Z 849.669,A -85,B 0,C 180,E1 21851.514,E2 21851.514} C_VEL
LIN {X 0,Y 467.718,Z 834.206,A -85,B 0,C 180,E1 21849.902,E2 21849.902} C_VEL
LIN {X 0,Y 468.702,Z 818.587,A -85,B 0,C 180,E1 21848.559,E2 21848.559} C_VEL
LIN {X 0,Y 469.749,Z 802.172,A -85,B 0,C 180,E1 21847.407,E2 21847.407} C_VEL
LIN {X 0,Y 470.729,Z 784.415,A -85,B 0,C 180,E1 21846.416,E2 21846.416} C_VEL
LIN {X 0,Y 471.602,Z 766.248,A -85,B 0,C 180,E1 21845.647,E2 21845.647} C_VEL
LIN {X 0,Y 472.336,Z 747.45,A -85,B 0,C 180,E1 21845.091,E2 21845.091} C_VEL
LIN {X 0,Y 472.752,Z 722.173,A -85,B 0,C 180,E1 21844.646,E2 21844.646} C_VEL
LIN {X 0,Y 474.33,Z 556.216,A -85,B 0,C 180,E1 21842.091,E2 21842.091} C_VEL
LIN {X 0,Y 472.382,Z 539.766,A -85,B 0,C 180,E1 21841.681,E2 21841.681} C_VEL
LIN {X 0,Y 475.222,Z 495.688,A -85,B 0,C 180,E1 21837.839,E2 21837.839} C_VEL
LIN {X 0,Y 476.496,Z 477.499,A -85,B 0,C 180,E1 21836.196,E2 21836.196} C_VEL
LIN {X 0,Y 470.137,Z 458.801,A -85,B 0,C 180,E1 21833.813,E2 21833.813} C_VEL
LIN {X 0,Y 465.047,Z 445.172,A -85,B 0,C 180,E1 21831.864,E2 21831.864} C_VEL
LIN {X 0,Y 465.013,Z 444.874,A -85,B 0,C 180,E1 21830.14,E2 21830.14} C_VEL
LIN {X 0,Y 465.008,Z 444.872,A -85,B 0,C 180,E1 21826.437,E2 21826.437} C_VEL
LIN {X 0,Y 465.008,Z 444.871,A -85,B 0,C 180,E1 21822.662,E2 21822.662} C_VEL
LIN {X 0,Y 465.009,Z 444.864,A -85,B 0,C 180,E1 21819.05,E2 21819.05} C_VEL
LIN {X 0,Y 464.998,Z 444.87,A -85,B 0,C 180,E1 21815.339,E2 21815.339} C_VEL
LIN {X 0,Y 465.006,Z 444.868,A -85,B 0,C 180,E1 21811.627,E2 21811.627} C_VEL
LIN {X 0,Y 465.011,Z 444.863,A -85,B 0,C 180,E1 21807.952,E2 21807.952} C_VEL
LIN {X 0,Y 465.008,Z 444.864,A -85,B 0,C 180,E1 21804.248,E2 21804.248} C_VEL
LIN {X 0,Y 465.007,Z 444.868,A -85,B 0,C 180,E1 21800.648,E2 21800.648} C_VEL
LIN {X 0,Y 464.999,Z 444.874,A -85,B 0,C 180,E1 21797.003,E2 21797.003} C_VEL
LIN {X 0,Y 465.008,Z 444.868,A -85,B 0,C 180,E1 21793.301,E2 21793.301} C_VEL
LIN {X 0,Y 465.008,Z 444.861,A -85,B 0,C 180,E1 21789.655,E2 21789.655} C_VEL
LIN {X 0,Y 465.012,Z 444.87,A -85,B 0,C 180,E1 21785.924,E2 21785.924} C_VEL
LIN {X 0,Y 465.005,Z 444.872,A -85,B 0,C 180,E1 21782.218,E2 21782.218} C_VEL
LIN {X 0,Y 464.996,Z 444.873,A -85,B 0,C 180,E1 21778.521,E2 21778.521} C_VEL
LIN {X 0,Y 465.001,Z 444.863,A -85,B 0,C 180,E1 21774.818,E2 21774.818} C_VEL
LIN {X 0,Y 465.01,Z 444.867,A -85,B 0,C 180,E1 21771.218,E2 21771.218} C_VEL
LIN {X 0,Y 465.01,Z 444.872,A -85,B 0,C 180,E1 21767.457,E2 21767.457} C_VEL
LIN {X 0,Y 465.008,Z 444.872,A -85,B 0,C 180,E1 21763.768,E2 21763.768} C_VEL
LIN {X 0,Y 464.993,Z 444.874,A -85,B 0,C 180,E1 21760.139,E2 21760.139} C_VEL
LIN {X 0,Y 465.003,Z 444.871,A -85,B 0,C 180,E1 21756.425,E2 21756.425} C_VEL
LIN {X 0,Y 465.012,Z 444.869,A -85,B 0,C 180,E1 21752.742,E2 21752.742} C_VEL
LIN {X 0,Y 465.014,Z 444.874,A -85,B 0,C 180,E1 21749.076,E2 21749.076} C_VEL
LIN {X 0,Y 465.002,Z 444.872,A -85,B 0,C 180,E1 21745.412,E2 21745.412} C_VEL
LIN {X 0,Y 465.032,Z 445.156,A -85,B 0,C 180,E1 21743.886,E2 21743.886} C_VEL
LIN {X 0,Y 470.033,Z 461.326,A -85,B 0,C 180,E1 21740.975,E2 21740.975} C_VEL
LIN {X 0,Y 473.014,Z 472.835,A -85,B 0,C 180,E1 21739.059,E2 21739.059} C_VEL
LIN {X 0,Y 470.97,Z 501.011,A -85,B 0,C 180,E1 21735.237,E2 21735.237} C_VEL
LIN {X 0,Y 469.254,Z 529.811,A -85,B 0,C 180,E1 21731.407,E2 21731.407} C_VEL
LIN {X 0,Y 467.921,Z 555.21,A -85,B 0,C 180,E1 21728.098,E2 21728.098} C_VEL
LIN {X 0,Y 470.931,Z 571.678,A -85,B 0,C 180,E1 21727.618,E2 21727.618} C_VEL
LIN {X 0,Y 470.418,Z 621.736,A -85,B 0,C 180,E1 21726.808,E2 21726.808} C_VEL
LIN {X 0,Y 469.408,Z 629.408,A -85,B 0,C 180,E1 21726.731,E2 21726.731} C_VEL
LIN {X 0,Y 463.368,Z 649.778,A -85,B 0,C 180,E1 21726.693,E2 21726.693} C_VEL
LIN {X 0,Y 462.565,Z 656.362,A -85,B 0,C 180,E1 21726.618,E2 21726.618} C_VEL
LIN {X 0,Y 462.25,Z 678.302,A -85,B 0,C 180,E1 21726.183,E2 21726.183} C_VEL
LIN {X 0,Y 461.865,Z 693.101,A -85,B 0,C 180,E1 21725.657,E2 21725.657} C_VEL
LIN {X 0,Y 461.285,Z 707.594,A -85,B 0,C 180,E1 21724.906,E2 21724.906} C_VEL
LIN {X 0,Y 460.527,Z 721.539,A -85,B 0,C 180,E1 21723.916,E2 21723.916} C_VEL
LIN {X 0,Y 459.755,Z 733.765,A -85,B 0,C 180,E1 21722.787,E2 21722.787} C_VEL
LIN {X 0,Y 459.027,Z 744.908,A -85,B 0,C 180,E1 21721.478,E2 21721.478} C_VEL
LIN {X 0,Y 458.31,Z 754.955,A -85,B 0,C 180,E1 21719.973,E2 21719.973} C_VEL
LIN {X 0,Y 457.752,Z 763.048,A -85,B 0,C 180,E1 21718.436,E2 21718.436} C_VEL
LIN {X 0,Y 457.249,Z 770.439,A -85,B 0,C 180,E1 21716.574,E2 21716.574} C_VEL
LIN {X 0,Y 456.918,Z 775.691,A -85,B 0,C 180,E1 21714.706,E2 21714.706} C_VEL
LIN {X 0,Y 456.728,Z 779.138,A -85,B 0,C 180,E1 21712.798,E2 21712.798} C_VEL
LIN {X 0,Y 456.639,Z 780.809,A -85,B 0,C 180,E1 21710.776,E2 21710.776} C_VEL
LIN {X 0,Y 456.629,Z 780.535,A -85,B 0,C 180,E1 21708.776,E2 21708.776} C_VEL
LIN {X 0,Y 456.703,Z 778.606,A -85,B 0,C 180,E1 21706.916,E2 21706.916} C_VEL
LIN {X 0,Y 456.885,Z 774.694,A -85,B 0,C 180,E1 21704.965,E2 21704.965} C_VEL
LIN {X 0,Y 457.188,Z 769.148,A -85,B 0,C 180,E1 21703.147,E2 21703.147} C_VEL
LIN {X 0,Y 457.62,Z 762.204,A -85,B 0,C 180,E1 21701.468,E2 21701.468} C_VEL
LIN {X 0,Y 458.196,Z 753.098,A -85,B 0,C 180,E1 21699.8,E2 21699.8} C_VEL
LIN {X 0,Y 458.84,Z 743.19,A -85,B 0,C 180,E1 21698.382,E2 21698.382} C_VEL
LIN {X 0,Y 459.567,Z 731.526,A -85,B 0,C 180,E1 21697.061,E2 21697.061} C_VEL
LIN {X 0,Y 460.303,Z 718.522,A -85,B 0,C 180,E1 21695.922,E2 21695.922} C_VEL
LIN {X 0,Y 460.939,Z 705.437,A -85,B 0,C 180,E1 21695.04,E2 21695.04} C_VEL
LIN {X 0,Y 461.509,Z 690.152,A -85,B 0,C 180,E1 21694.286,E2 21694.286} C_VEL
LIN {X 0,Y 461.87,Z 674.167,A -85,B 0,C 180,E1 21693.778,E2 21693.778} C_VEL
LIN {X 0,Y 462.894,Z 571.791,A -85,B 0,C 180,E1 21692.077,E2 21692.077} C_VEL
LIN {X 0,Y 459.967,Z 555.172,A -85,B 0,C 180,E1 21691.619,E2 21691.619} C_VEL
LIN {X 0,Y 461.418,Z 525.649,A -85,B 0,C 180,E1 21687.764,E2 21687.764} C_VEL
LIN {X 0,Y 463.179,Z 496.81,A -85,B 0,C 180,E1 21683.928,E2 21683.928} C_VEL
LIN {X 0,Y 464.705,Z 473.457,A -85,B 0,C 180,E1 21680.776,E2 21680.776} C_VEL
LIN {X 0,Y 459.977,Z 456.167,A -85,B 0,C 180,E1 21677.955,E2 21677.955} C_VEL
LIN {X 0,Y 457.034,Z 445.965,A -85,B 0,C 180,E1 21676.172,E2 21676.172} C_VEL
LIN {X 0,Y 457.004,Z 445.869,A -85,B 0,C 180,E1 21672.537,E2 21672.537} C_VEL
LIN {X 0,Y 457.011,Z 445.867,A -85,B 0,C 180,E1 21668.839,E2 21668.839} C_VEL
LIN {X 0,Y 457.047,Z 445.846,A -85,B 0,C 180,E1 21665.301,E2 21665.301} C_VEL
LIN {X 0,Y 457.031,Z 445.861,A -85,B 0,C 180,E1 21661.658,E2 21661.658} C_VEL
LIN {X 0,Y 456.995,Z 445.864,A -85,B 0,C 180,E1 21658.178,E2 21658.178} C_VEL
LIN {X 0,Y 456.999,Z 445.866,A -85,B 0,C 180,E1 21654.41,E2 21654.41} C_VEL
LIN {X 0,Y 457.028,Z 445.868,A -85,B 0,C 180,E1 21650.783,E2 21650.783} C_VEL
LIN {X 0,Y 457.044,Z 445.853,A -85,B 0,C 180,E1 21647.298,E2 21647.298} C_VEL
LIN {X 0,Y 457.011,Z 445.868,A -85,B 0,C 180,E1 21643.738,E2 21643.738} C_VEL
LIN {X 0,Y 457.008,Z 445.86,A -85,B 0,C 180,E1 21640.026,E2 21640.026} C_VEL
LIN {X 0,Y 457.037,Z 445.86,A -85,B 0,C 180,E1 21636.517,E2 21636.517} C_VEL
LIN {X 0,Y 457.063,Z 445.851,A -85,B 0,C 180,E1 21632.856,E2 21632.856} C_VEL
LIN {X 0,Y 457.028,Z 445.867,A -85,B 0,C 180,E1 21629.345,E2 21629.345} C_VEL
LIN {X 0,Y 457.015,Z 445.844,A -85,B 0,C 180,E1 21625.67,E2 21625.67} C_VEL
LIN {X 0,Y 457.027,Z 445.865,A -85,B 0,C 180,E1 21621.969,E2 21621.969} C_VEL
LIN {X 0,Y 457.059,Z 445.838,A -85,B 0,C 180,E1 21618.362,E2 21618.362} C_VEL
LIN {X 0,Y 457.069,Z 445.859,A -85,B 0,C 180,E1 21614.7,E2 21614.7} C_VEL
LIN {X 0,Y 457.034,Z 445.863,A -85,B 0,C 180,E1 21611.1,E2 21611.1} C_VEL
LIN {X 0,Y 457.026,Z 445.849,A -85,B 0,C 180,E1 21607.417,E2 21607.417} C_VEL
LIN {X 0,Y 457.045,Z 445.861,A -85,B 0,C 180,E1 21603.763,E2 21603.763} C_VEL
LIN {X 0,Y 457.079,Z 445.838,A -85,B 0,C 180,E1 21600.126,E2 21600.126} C_VEL
LIN {X 0,Y 457.071,Z 445.866,A -85,B 0,C 180,E1 21596.363,E2 21596.363} C_VEL
LIN {X 0,Y 457.047,Z 445.849,A -85,B 0,C 180,E1 21592.711,E2 21592.711} C_VEL
LIN {X 0,Y 457.039,Z 445.863,A -85,B 0,C 180,E1 21589.028,E2 21589.028} C_VEL
LIN {X 0,Y 457.047,Z 445.847,A -85,B 0,C 180,E1 21585.3,E2 21585.3} C_VEL
LIN {X 0,Y 457.073,Z 445.861,A -85,B 0,C 180,E1 21581.639,E2 21581.639} C_VEL
LIN {X 0,Y 457.076,Z 445.851,A -85,B 0,C 180,E1 21577.898,E2 21577.898} C_VEL
LIN {X 0,Y 457.066,Z 445.858,A -85,B 0,C 180,E1 21574.194,E2 21574.194} C_VEL
LIN {X 0,Y 457.052,Z 445.865,A -85,B 0,C 180,E1 21570.514,E2 21570.514} C_VEL
LIN {X 0,Y 457.055,Z 445.86,A -85,B 0,C 180,E1 21566.845,E2 21566.845} C_VEL
LIN {X 0,Y 457.071,Z 445.86,A -85,B 0,C 180,E1 21563.174,E2 21563.174} C_VEL
LIN {X 0,Y 457.072,Z 445.864,A -85,B 0,C 180,E1 21559.481,E2 21559.481} C_VEL
LIN {X 0,Y 457.073,Z 445.864,A -85,B 0,C 180,E1 21555.748,E2 21555.748} C_VEL
LIN {X 0,Y 457.065,Z 445.86,A -85,B 0,C 180,E1 21552.021,E2 21552.021} C_VEL
LIN {X 0,Y 457.078,Z 445.989,A -85,B 0,C 180,E1 21548.328,E2 21548.328} C_VEL
LIN {X 0,Y 457.421,Z 447.425,A -85,B 0,C 180,E1 21548.055,E2 21548.055} C_VEL
LIN {X 0,Y 465.264,Z 469.278,A -85,B 0,C 180,E1 21545.252,E2 21545.252} C_VEL
LIN {X 0,Y 468.861,Z 480.599,A -85,B 0,C 180,E1 21543.901,E2 21543.901} C_VEL
LIN {X 0,Y 465.762,Z 524.544,A -85,B 0,C 180,E1 21540.012,E2 21540.012} C_VEL
LIN {X 0,Y 464.893,Z 540.548,A -85,B 0,C 180,E1 21538.658,E2 21538.658} C_VEL
LIN {X 0,Y 467.109,Z 560.28,A -85,B 0,C 180,E1 21538.218,E2 21538.218} C_VEL
LIN {X 0,Y 464.982,Z 742.822,A -85,B 0,C 180,E1 21535.361,E2 21535.361} C_VEL
LIN {X 0,Y 464.295,Z 761.63,A -85,B 0,C 180,E1 21534.848,E2 21534.848} C_VEL
LIN {X 0,Y 463.384,Z 779.946,A -85,B 0,C 180,E1 21534.116,E2 21534.116} C_VEL
LIN {X 0,Y 462.363,Z 797.521,A -85,B 0,C 180,E1 21533.177,E2 21533.177} C_VEL
LIN {X 0,Y 461.252,Z 814.49,A -85,B 0,C 180,E1 21532.025,E2 21532.025} C_VEL
LIN {X 0,Y 460.119,Z 831.257,A -85,B 0,C 180,E1 21530.612,E2 21530.612} C_VEL
LIN {X 0,Y 459.054,Z 846.525,A -85,B 0,C 180,E1 21529.041,E2 21529.041} C_VEL
LIN {X 0,Y 458.168,Z 859.811,A -85,B 0,C 180,E1 21527.396,E2 21527.396} C_VEL
LIN {X 0,Y 457.432,Z 871.987,A -85,B 0,C 180,E1 21525.596,E2 21525.596} C_VEL
LIN {X 0,Y 456.869,Z 882.86,A -85,B 0,C 180,E1 21523.665,E2 21523.665} C_VEL
LIN {X 0,Y 456.505,Z 892.301,A -85,B 0,C 180,E1 21521.625,E2 21521.625} C_VEL
LIN {X 0,Y 456.293,Z 900.348,A -85,B 0,C 180,E1 21519.459,E2 21519.459} C_VEL
LIN {X 0,Y 456.226,Z 906.545,A -85,B 0,C 180,E1 21517.303,E2 21517.303} C_VEL
LIN {X 0,Y 456.237,Z 911.267,A -85,B 0,C 180,E1 21515.029,E2 21515.029} C_VEL
LIN {X 0,Y 456.271,Z 914.196,A -85,B 0,C 180,E1 21512.764,E2 21512.764} C_VEL
LIN {X 0,Y 456.295,Z 915.403,A -85,B 0,C 180,E1 21510.502,E2 21510.502} C_VEL
LIN {X 0,Y 456.293,Z 914.914,A -85,B 0,C 180,E1 21508.242,E2 21508.242} C_VEL
LIN {X 0,Y 456.268,Z 912.719,A -85,B 0,C 180,E1 21505.979,E2 21505.979} C_VEL
LIN {X 0,Y 456.242,Z 908.769,A -85,B 0,C 180,E1 21503.709,E2 21503.709} C_VEL
LIN {X 0,Y 456.262,Z 902.964,A -85,B 0,C 180,E1 21501.43,E2 21501.43} C_VEL
LIN {X 0,Y 456.423,Z 895.162,A -85,B 0,C 180,E1 21499.141,E2 21499.141} C_VEL
LIN {X 0,Y 456.719,Z 886.348,A -85,B 0,C 180,E1 21497.097,E2 21497.097} C_VEL
LIN {X 0,Y 457.218,Z 875.512,A -85,B 0,C 180,E1 21495.046,E2 21495.046} C_VEL
LIN {X 0,Y 457.927,Z 863.167,A -85,B 0,C 180,E1 21493.118,E2 21493.118} C_VEL
LIN {X 0,Y 458.816,Z 849.253,A -85,B 0,C 180,E1 21491.316,E2 21491.316} C_VEL
LIN {X 0,Y 459.857,Z 834.274,A -85,B 0,C 180,E1 21489.709,E2 21489.709} C_VEL
LIN {X 0,Y 460.934,Z 818.313,A -85,B 0,C 180,E1 21488.298,E2 21488.298} C_VEL
LIN {X 0,Y 462.086,Z 801.241,A -85,B 0,C 180,E1 21487.078,E2 21487.078} C_VEL
LIN {X 0,Y 463.123,Z 783.774,A -85,B 0,C 180,E1 21486.088,E2 21486.088} C_VEL
LIN {X 0,Y 464.055,Z 765.568,A -85,B 0,C 180,E1 21485.305,E2 21485.305} C_VEL
LIN {X 0,Y 464.827,Z 746.869,A -85,B 0,C 180,E1 21484.744,E2 21484.744} C_VEL
LIN {X 0,Y 465.261,Z 722.77,A -85,B 0,C 180,E1 21484.308,E2 21484.308} C_VEL
LIN {X 0,Y 466.999,Z 557.206,A -85,B 0,C 180,E1 21481.711,E2 21481.711} C_VEL
LIN {X 0,Y 464.973,Z 539.989,A -85,B 0,C 180,E1 21481.275,E2 21481.275} C_VEL
LIN {X 0,Y 468.018,Z 496.761,A -85,B 0,C 180,E1 21477.428,E2 21477.428} C_VEL
LIN {X 0,Y 469.295,Z 480.388,A -85,B 0,C 180,E1 21475.921,E2 21475.921} C_VEL
LIN {X 0,Y 462.941,Z 461.544,A -85,B 0,C 180,E1 21473.46,E2 21473.46} C_VEL
LIN {X 0,Y 457.104,Z 446.066,A -85,B 0,C 180,E1 21471.155,E2 21471.155} C_VEL
LIN {X 0,Y 457.063,Z 445.858,A -85,B 0,C 180,E1 21467.494,E2 21467.494} C_VEL
LIN {X 0,Y 457.066,Z 445.866,A -85,B 0,C 180,E1 21463.73,E2 21463.73} C_VEL
LIN {X 0,Y 457.073,Z 445.86,A -85,B 0,C 180,E1 21460.026,E2 21460.026} C_VEL
LIN {X 0,Y 457.067,Z 445.858,A -85,B 0,C 180,E1 21456.358,E2 21456.358} C_VEL
LIN {X 0,Y 457.072,Z 445.855,A -85,B 0,C 180,E1 21452.627,E2 21452.627} C_VEL
LIN {X 0,Y 457.066,Z 445.854,A -85,B 0,C 180,E1 21448.911,E2 21448.911} C_VEL
LIN {X 0,Y 457.061,Z 445.858,A -85,B 0,C 180,E1 21445.25,E2 21445.25} C_VEL
LIN {X 0,Y 457.075,Z 445.865,A -85,B 0,C 180,E1 21441.561,E2 21441.561} C_VEL
LIN {X 0,Y 457.069,Z 445.858,A -85,B 0,C 180,E1 21437.834,E2 21437.834} C_VEL
LIN {X 0,Y 457.073,Z 445.845,A -85,B 0,C 180,E1 21434.182,E2 21434.182} C_VEL
LIN {X 0,Y 457.064,Z 445.853,A -85,B 0,C 180,E1 21430.461,E2 21430.461} C_VEL
LIN {X 0,Y 457.056,Z 445.863,A -85,B 0,C 180,E1 21426.784,E2 21426.784} C_VEL
LIN {X 0,Y 457.069,Z 445.858,A -85,B 0,C 180,E1 21423.135,E2 21423.135} C_VEL
LIN {X 0,Y 457.07,Z 445.848,A -85,B 0,C 180,E1 21419.498,E2 21419.498} C_VEL
LIN {X 0,Y 457.071,Z 445.856,A -85,B 0,C 180,E1 21415.734,E2 21415.734} C_VEL
LIN {X 0,Y 457.062,Z 445.86,A -85,B 0,C 180,E1 21412.078,E2 21412.078} C_VEL
LIN {X 0,Y 457.056,Z 445.864,A -85,B 0,C 180,E1 21408.389,E2 21408.389} C_VEL
LIN {X 0,Y 457.067,Z 445.864,A -85,B 0,C 180,E1 21404.651,E2 21404.651} C_VEL
LIN {X 0,Y 457.072,Z 445.861,A -85,B 0,C 180,E1 21400.911,E2 21400.911} C_VEL
LIN {X 0,Y 457.075,Z 445.862,A -85,B 0,C 180,E1 21397.22,E2 21397.22} C_VEL
LIN {X 0,Y 457.071,Z 445.862,A -85,B 0,C 180,E1 21393.47,E2 21393.47} C_VEL
LIN {X 0,Y 457.055,Z 445.86,A -85,B 0,C 180,E1 21389.781,E2 21389.781} C_VEL
LIN {X 0,Y 457.055,Z 445.862,A -85,B 0,C 180,E1 21386.006,E2 21386.006} C_VEL
LIN {X 0,Y 457.117,Z 446.178,A -85,B 0,C 180,E1 21384.527,E2 21384.527} C_VEL
LIN {X 0,Y 461.845,Z 461.142,A -85,B 0,C 180,E1 21381.744,E2 21381.744} C_VEL
LIN {X 0,Y 465.65,Z 475.445,A -85,B 0,C 180,E1 21379.286,E2 21379.286} C_VEL
LIN {X 0,Y 463.505,Z 503.059,A -85,B 0,C 180,E1 21375.486,E2 21375.486} C_VEL
LIN {X 0,Y 461.659,Z 531.851,A -85,B 0,C 180,E1 21371.6,E2 21371.6} C_VEL
LIN {X 0,Y 460.373,Z 555.263,A -85,B 0,C 180,E1 21368.523,E2 21368.523} C_VEL
LIN {X 0,Y 463.753,Z 574.342,A -85,B 0,C 180,E1 21367.972,E2 21367.972} C_VEL
LIN {X 0,Y 462.565,Z 656.362,A -85,B 0,C 180,E1 21366.618,E2 21366.618} C_VEL
LIN {X 0,Y 461.484,Z 664.035,A -85,B 0,C 180,E1 21366.542,E2 21366.542} C_VEL
LIN {X 0,Y 456.124,Z 681.072,A -85,B 0,C 180,E1 21366.424,E2 21366.424} C_VEL
LIN {X 0,Y 454.683,Z 688.591,A -85,B 0,C 180,E1 21366.232,E2 21366.232} C_VEL
LIN {X 0,Y 454.55,Z 690.652,A -85,B 0,C 180,E1 21366.155,E2 21366.155} C_VEL
LIN {X 0,Y 453.996,Z 704.654,A -85,B 0,C 180,E1 21365.473,E2 21365.473} C_VEL
LIN {X 0,Y 453.246,Z 718.748,A -85,B 0,C 180,E1 21364.537,E2 21364.537} C_VEL
LIN {X 0,Y 452.374,Z 731.779,A -85,B 0,C 180,E1 21363.391,E2 21363.391} C_VEL
LIN {X 0,Y 451.578,Z 743.246,A -85,B 0,C 180,E1 21362.1,E2 21362.1} C_VEL
LIN {X 0,Y 450.785,Z 753.637,A -85,B 0,C 180,E1 21360.615,E2 21360.615} C_VEL
LIN {X 0,Y 450.09,Z 762.618,A -85,B 0,C 180,E1 21358.965,E2 21358.965} C_VEL
LIN {X 0,Y 449.556,Z 769.745,A -85,B 0,C 180,E1 21357.269,E2 21357.269} C_VEL
LIN {X 0,Y 449.125,Z 775.725,A -85,B 0,C 180,E1 21355.305,E2 21355.305} C_VEL
LIN {X 0,Y 448.87,Z 779.608,A -85,B 0,C 180,E1 21353.359,E2 21353.359} C_VEL
LIN {X 0,Y 448.748,Z 781.686,A -85,B 0,C 180,E1 21351.433,E2 21351.433} C_VEL
LIN {X 0,Y 448.709,Z 781.988,A -85,B 0,C 180,E1 21349.391,E2 21349.391} C_VEL
LIN {X 0,Y 448.76,Z 780.6,A -85,B 0,C 180,E1 21347.505,E2 21347.505} C_VEL
LIN {X 0,Y 448.922,Z 777.306,A -85,B 0,C 180,E1 21345.502,E2 21345.502} C_VEL
LIN {X 0,Y 449.198,Z 772.382,A -85,B 0,C 180,E1 21343.647,E2 21343.647} C_VEL
LIN {X 0,Y 449.616,Z 765.999,A -85,B 0,C 180,E1 21341.908,E2 21341.908} C_VEL
LIN {X 0,Y 450.221,Z 757.139,A -85,B 0,C 180,E1 21340.104,E2 21340.104} C_VEL
LIN {X 0,Y 450.922,Z 746.999,A -85,B 0,C 180,E1 21338.525,E2 21338.525} C_VEL
LIN {X 0,Y 451.662,Z 736.096,A -85,B 0,C 180,E1 21337.185,E2 21337.185} C_VEL
LIN {X 0,Y 452.447,Z 723.401,A -85,B 0,C 180,E1 21335.962,E2 21335.962} C_VEL
LIN {X 0,Y 453.145,Z 710.619,A -85,B 0,C 180,E1 21335.012,E2 21335.012} C_VEL
LIN {X 0,Y 453.775,Z 696.162,A -85,B 0,C 180,E1 21334.201,E2 21334.201} C_VEL
LIN {X 0,Y 454.24,Z 680.061,A -85,B 0,C 180,E1 21333.589,E2 21333.589} C_VEL
LIN {X 0,Y 454.494,Z 662.757,A -85,B 0,C 180,E1 21333.216,E2 21333.216} C_VEL
LIN {X 0,Y 455.461,Z 572.916,A -85,B 0,C 180,E1 21331.726,E2 21331.726} C_VEL
LIN {X 0,Y 452.356,Z 555.608,A -85,B 0,C 180,E1 21331.266,E2 21331.266} C_VEL
LIN {X 0,Y 452.472,Z 551.305,A -85,B 0,C 180,E1 21330.759,E2 21330.759} C_VEL
LIN {X 0,Y 454.191,Z 521.065,A -85,B 0,C 180,E1 21326.719,E2 21326.719} C_VEL
LIN {X 0,Y 455.998,Z 493.171,A -85,B 0,C 180,E1 21322.947,E2 21322.947} C_VEL
LIN {X 0,Y 457.152,Z 475.671,A -85,B 0,C 180,E1 21320.544,E2 21320.544} C_VEL
LIN {X 0,Y 452.101,Z 457.21,A -85,B 0,C 180,E1 21317.482,E2 21317.482} C_VEL
LIN {X 0,Y 449.142,Z 446.967,A -85,B 0,C 180,E1 21315.661,E2 21315.661} C_VEL
LIN {X 0,Y 449.091,Z 446.858,A -85,B 0,C 180,E1 21311.931,E2 21311.931} C_VEL
LIN {X 0,Y 449.064,Z 446.849,A -85,B 0,C 180,E1 21308.308,E2 21308.308} C_VEL
LIN {X 0,Y 449.061,Z 446.856,A -85,B 0,C 180,E1 21304.55,E2 21304.55} C_VEL
LIN {X 0,Y 449.082,Z 446.855,A -85,B 0,C 180,E1 21300.963,E2 21300.963} C_VEL
LIN {X 0,Y 449.113,Z 446.846,A -85,B 0,C 180,E1 21297.304,E2 21297.304} C_VEL
LIN {X 0,Y 449.078,Z 446.85,A -85,B 0,C 180,E1 21293.683,E2 21293.683} C_VEL
LIN {X 0,Y 449.062,Z 446.858,A -85,B 0,C 180,E1 21290.115,E2 21290.115} C_VEL
LIN {X 0,Y 449.078,Z 446.853,A -85,B 0,C 180,E1 21286.529,E2 21286.529} C_VEL
LIN {X 0,Y 449.117,Z 446.843,A -85,B 0,C 180,E1 21282.908,E2 21282.908} C_VEL
LIN {X 0,Y 449.091,Z 446.85,A -85,B 0,C 180,E1 21279.385,E2 21279.385} C_VEL
LIN {X 0,Y 449.071,Z 446.849,A -85,B 0,C 180,E1 21275.844,E2 21275.844} C_VEL
LIN {X 0,Y 449.082,Z 446.851,A -85,B 0,C 180,E1 21272.149,E2 21272.149} C_VEL
LIN {X 0,Y 449.126,Z 446.844,A -85,B 0,C 180,E1 21268.597,E2 21268.597} C_VEL
LIN {X 0,Y 449.119,Z 446.835,A -85,B 0,C 180,E1 21264.883,E2 21264.883} C_VEL
LIN {X 0,Y 449.09,Z 446.855,A -85,B 0,C 180,E1 21261.279,E2 21261.279} C_VEL
LIN {X 0,Y 449.082,Z 446.827,A -85,B 0,C 180,E1 21257.626,E2 21257.626} C_VEL
LIN {X 0,Y 449.108,Z 446.851,A -85,B 0,C 180,E1 21254.044,E2 21254.044} C_VEL
LIN {X 0,Y 449.133,Z 446.834,A -85,B 0,C 180,E1 21250.389,E2 21250.389} C_VEL
LIN {X 0,Y 449.123,Z 446.84,A -85,B 0,C 180,E1 21246.648,E2 21246.648} C_VEL
LIN {X 0,Y 449.101,Z 446.853,A -85,B 0,C 180,E1 21242.935,E2 21242.935} C_VEL
LIN {X 0,Y 449.092,Z 446.834,A -85,B 0,C 180,E1 21239.235,E2 21239.235} C_VEL
LIN {X 0,Y 449.107,Z 446.851,A -85,B 0,C 180,E1 21235.531,E2 21235.531} C_VEL
LIN {X 0,Y 449.135,Z 446.83,A -85,B 0,C 180,E1 21231.938,E2 21231.938} C_VEL
LIN {X 0,Y 449.135,Z 446.853,A -85,B 0,C 180,E1 21228.182,E2 21228.182} C_VEL
LIN {X 0,Y 449.115,Z 446.835,A -85,B 0,C 180,E1 21224.505,E2 21224.505} C_VEL
LIN {X 0,Y 449.108,Z 446.853,A -85,B 0,C 180,E1 21220.762,E2 21220.762} C_VEL
LIN {X 0,Y 449.11,Z 446.847,A -85,B 0,C 180,E1 21216.932,E2 21216.932} C_VEL
LIN {X 0,Y 449.124,Z 446.837,A -85,B 0,C 180,E1 21213.218,E2 21213.218} C_VEL
LIN {X 0,Y 449.139,Z 446.845,A -85,B 0,C 180,E1 21209.489,E2 21209.489} C_VEL
LIN {X 0,Y 449.135,Z 446.85,A -85,B 0,C 180,E1 21205.682,E2 21205.682} C_VEL
LIN {X 0,Y 449.134,Z 446.853,A -85,B 0,C 180,E1 21201.928,E2 21201.928} C_VEL
LIN {X 0,Y 449.121,Z 446.852,A -85,B 0,C 180,E1 21198.228,E2 21198.228} C_VEL
LIN {X 0,Y 449.12,Z 446.847,A -85,B 0,C 180,E1 21194.53,E2 21194.53} C_VEL
LIN {X 0,Y 449.136,Z 446.853,A -85,B 0,C 180,E1 21190.808,E2 21190.808} C_VEL
LIN {X 0,Y 449.18,Z 447.155,A -85,B 0,C 180,E1 21188.823,E2 21188.823} C_VEL
LIN {X 0,Y 457.475,Z 470.622,A -85,B 0,C 180,E1 21185.701,E2 21185.701} C_VEL
LIN {X 0,Y 461.532,Z 482.764,A -85,B 0,C 180,E1 21184.207,E2 21184.207} C_VEL
LIN {X 0,Y 458.239,Z 526.499,A -85,B 0,C 180,E1 21180.267,E2 21180.267} C_VEL
LIN {X 0,Y 457.384,Z 540.244,A -85,B 0,C 180,E1 21179.065,E2 21179.065} C_VEL
LIN {X 0,Y 459.686,Z 561.177,A -85,B 0,C 180,E1 21178.578,E2 21178.578} C_VEL
LIN {X 0,Y 457.468,Z 742.368,A -85,B 0,C 180,E1 21175.708,E2 21175.708} C_VEL
LIN {X 0,Y 456.743,Z 761.185,A -85,B 0,C 180,E1 21175.187,E2 21175.187} C_VEL
LIN {X 0,Y 455.831,Z 778.457,A -85,B 0,C 180,E1 21174.492,E2 21174.492} C_VEL
LIN {X 0,Y 454.734,Z 796.418,A -85,B 0,C 180,E1 21173.525,E2 21173.525} C_VEL
LIN {X 0,Y 453.559,Z 813.481,A -85,B 0,C 180,E1 21172.351,E2 21172.351} C_VEL
LIN {X 0,Y 452.345,Z 830.261,A -85,B 0,C 180,E1 21170.915,E2 21170.915} C_VEL
LIN {X 0,Y 451.237,Z 845.282,A -85,B 0,C 180,E1 21169.346,E2 21169.346} C_VEL
LIN {X 0,Y 450.245,Z 859.302,A -85,B 0,C 180,E1 21167.579,E2 21167.579} C_VEL
LIN {X 0,Y 449.431,Z 872.2,A -85,B 0,C 180,E1 21165.616,E2 21165.616} C_VEL
LIN {X 0,Y 448.84,Z 883.485,A -85,B 0,C 180,E1 21163.527,E2 21163.527} C_VEL
LIN {X 0,Y 448.479,Z 893.143,A -85,B 0,C 180,E1 21161.315,E2 21161.315} C_VEL
LIN {X 0,Y 448.3,Z 900.771,A -85,B 0,C 180,E1 21159.112,E2 21159.112} C_VEL
LIN {X 0,Y 448.268,Z 906.596,A -85,B 0,C 180,E1 21156.918,E2 21156.918} C_VEL
LIN {X 0,Y 448.307,Z 910.929,A -85,B 0,C 180,E1 21154.606,E2 21154.606} C_VEL
LIN {X 0,Y 448.356,Z 913.488,A -85,B 0,C 180,E1 21152.301,E2 21152.301} C_VEL
LIN {X 0,Y 448.386,Z 914.324,A -85,B 0,C 180,E1 21150,E2 21150} C_VEL
LIN {X 0,Y 448.363,Z 913.443,A -85,B 0,C 180,E1 21147.7,E2 21147.7} C_VEL
LIN {X 0,Y 448.318,Z 910.84,A -85,B 0,C 180,E1 21145.395,E2 21145.395} C_VEL
LIN {X 0,Y 448.281,Z 906.464,A -85,B 0,C 180,E1 21143.083,E2 21143.083} C_VEL
LIN {X 0,Y 448.32,Z 900.209,A -85,B 0,C 180,E1 21140.76,E2 21140.76} C_VEL
LIN {X 0,Y 448.504,Z 892.421,A -85,B 0,C 180,E1 21138.556,E2 21138.556} C_VEL
LIN {X 0,Y 448.871,Z 882.561,A -85,B 0,C 180,E1 21136.343,E2 21136.343} C_VEL
LIN {X 0,Y 449.477,Z 871.094,A -85,B 0,C 180,E1 21134.253,E2 21134.253} C_VEL
LIN {X 0,Y 450.264,Z 858.491,A -85,B 0,C 180,E1 21132.356,E2 21132.356} C_VEL
LIN {X 0,Y 451.257,Z 844.357,A -85,B 0,C 180,E1 21130.588,E2 21130.588} C_VEL
LIN {X 0,Y 452.409,Z 828.581,A -85,B 0,C 180,E1 21128.959,E2 21128.959} C_VEL
LIN {X 0,Y 453.597,Z 812.289,A -85,B 0,C 180,E1 21127.583,E2 21127.583} C_VEL
LIN {X 0,Y 454.783,Z 795.171,A -85,B 0,C 180,E1 21126.414,E2 21126.414} C_VEL
LIN {X 0,Y 455.862,Z 777.668,A -85,B 0,C 180,E1 21125.475,E2 21125.475} C_VEL
LIN {X 0,Y 456.853,Z 759.135,A -85,B 0,C 180,E1 21124.737,E2 21124.737} C_VEL
LIN {X 0,Y 457.58,Z 739.898,A -85,B 0,C 180,E1 21124.225,E2 21124.225} C_VEL
LIN {X 0,Y 459.691,Z 558.165,A -85,B 0,C 180,E1 21121.317,E2 21121.317} C_VEL
LIN {X 0,Y 457.589,Z 540.235,A -85,B 0,C 180,E1 21120.859,E2 21120.859} C_VEL
LIN {X 0,Y 460.905,Z 497.081,A -85,B 0,C 180,E1 21116.935,E2 21116.935} C_VEL
LIN {X 0,Y 462.041,Z 483.065,A -85,B 0,C 180,E1 21115.611,E2 21115.611} C_VEL
LIN {X 0,Y 456.116,Z 465.383,A -85,B 0,C 180,E1 21113.241,E2 21113.241} C_VEL
LIN {X 0,Y 450.007,Z 449.629,A -85,B 0,C 180,E1 21110.875,E2 21110.875} C_VEL
LIN {X 0,Y 449.156,Z 447.03,A -85,B 0,C 180,E1 21110.416,E2 21110.416} C_VEL
LIN {X 0,Y 449.13,Z 446.847,A -85,B 0,C 180,E1 21106.712,E2 21106.712} C_VEL
LIN {X 0,Y 449.133,Z 446.85,A -85,B 0,C 180,E1 21102.911,E2 21102.911} C_VEL
LIN {X 0,Y 449.125,Z 446.842,A -85,B 0,C 180,E1 21099.216,E2 21099.216} C_VEL
LIN {X 0,Y 449.121,Z 446.846,A -85,B 0,C 180,E1 21095.432,E2 21095.432} C_VEL
LIN {X 0,Y 449.13,Z 446.843,A -85,B 0,C 180,E1 21091.694,E2 21091.694} C_VEL
LIN {X 0,Y 449.131,Z 446.839,A -85,B 0,C 180,E1 21088.017,E2 21088.017} C_VEL
LIN {X 0,Y 449.13,Z 446.84,A -85,B 0,C 180,E1 21084.321,E2 21084.321} C_VEL
LIN {X 0,Y 449.132,Z 446.846,A -85,B 0,C 180,E1 21080.594,E2 21080.594} C_VEL
LIN {X 0,Y 449.123,Z 446.851,A -85,B 0,C 180,E1 21076.807,E2 21076.807} C_VEL
LIN {X 0,Y 449.121,Z 446.852,A -85,B 0,C 180,E1 21072.994,E2 21072.994} C_VEL
LIN {X 0,Y 449.127,Z 446.839,A -85,B 0,C 180,E1 21069.223,E2 21069.223} C_VEL
LIN {X 0,Y 449.13,Z 446.842,A -85,B 0,C 180,E1 21065.493,E2 21065.493} C_VEL
LIN {X 0,Y 449.132,Z 446.851,A -85,B 0,C 180,E1 21061.696,E2 21061.696} C_VEL
LIN {X 0,Y 449.131,Z 446.848,A -85,B 0,C 180,E1 21057.958,E2 21057.958} C_VEL
LIN {X 0,Y 449.119,Z 446.844,A -85,B 0,C 180,E1 21054.25,E2 21054.25} C_VEL
LIN {X 0,Y 449.117,Z 446.84,A -85,B 0,C 180,E1 21050.483,E2 21050.483} C_VEL
LIN {X 0,Y 449.129,Z 446.841,A -85,B 0,C 180,E1 21046.744,E2 21046.744} C_VEL
LIN {X 0,Y 449.133,Z 446.846,A -85,B 0,C 180,E1 21043.044,E2 21043.044} C_VEL
LIN {X 0,Y 449.134,Z 446.846,A -85,B 0,C 180,E1 21039.228,E2 21039.228} C_VEL
LIN {X 0,Y 449.13,Z 446.842,A -85,B 0,C 180,E1 21035.539,E2 21035.539} C_VEL
LIN {X 0,Y 449.118,Z 446.852,A -85,B 0,C 180,E1 21031.836,E2 21031.836} C_VEL
LIN {X 0,Y 449.117,Z 446.849,A -85,B 0,C 180,E1 21028.017,E2 21028.017} C_VEL
LIN {X 0,Y 449.172,Z 447.131,A -85,B 0,C 180,E1 21025.224,E2 21025.224} C_VEL
LIN {X 0,Y 454.112,Z 462.575,A -85,B 0,C 180,E1 21022.258,E2 21022.258} C_VEL
LIN {X 0,Y 458.293,Z 478.061,A -85,B 0,C 180,E1 21019.529,E2 21019.529} C_VEL
LIN {X 0,Y 456.048,Z 505.393,A -85,B 0,C 180,E1 21015.711,E2 21015.711} C_VEL
LIN {X 0,Y 454.108,Z 533.605,A -85,B 0,C 180,E1 21011.847,E2 21011.847} C_VEL
LIN {X 0,Y 452.83,Z 554.927,A -85,B 0,C 180,E1 21008.992,E2 21008.992} C_VEL
LIN {X 0,Y 454.198,Z 562.322,A -85,B 0,C 180,E1 21008.735,E2 21008.735} C_VEL
LIN {X 0,Y 456.459,Z 575.976,A -85,B 0,C 180,E1 21008.362,E2 21008.362} C_VEL
LIN {X 0,Y 454.927,Z 675.154,A -85,B 0,C 180,E1 21006.657,E2 21006.657} C_VEL
LIN {X 0,Y 454.55,Z 690.652,A -85,B 0,C 180,E1 21006.155,E2 21006.155} C_VEL
LIN {X 0,Y 453.391,Z 698.03,A -85,B 0,C 180,E1 21005.882,E2 21005.882} C_VEL
LIN {X 0,Y 448.255,Z 712.122,A -85,B 0,C 180,E1 21005.309,E2 21005.309} C_VEL
LIN {X 0,Y 445.924,Z 719.909,A -85,B 0,C 180,E1 21004.846,E2 21004.846} C_VEL
LIN {X 0,Y 445.542,Z 722.708,A -85,B 0,C 180,E1 21004.628,E2 21004.628} C_VEL
LIN {X 0,Y 444.649,Z 735.122,A -85,B 0,C 180,E1 21003.462,E2 21003.462} C_VEL
LIN {X 0,Y 443.777,Z 746.477,A -85,B 0,C 180,E1 21002.096,E2 21002.096} C_VEL
LIN {X 0,Y 442.994,Z 755.91,A -85,B 0,C 180,E1 21000.67,E2 21000.67} C_VEL
LIN {X 0,Y 442.242,Z 764.902,A -85,B 0,C 180,E1 20998.936,E2 20998.936} C_VEL
LIN {X 0,Y 441.635,Z 772.179,A -85,B 0,C 180,E1 20997.069,E2 20997.069} C_VEL
LIN {X 0,Y 441.228,Z 777.435,A -85,B 0,C 180,E1 20995.215,E2 20995.215} C_VEL
LIN {X 0,Y 440.951,Z 781.31,A -85,B 0,C 180,E1 20993.096,E2 20993.096} C_VEL
LIN {X 0,Y 440.82,Z 783.083,A -85,B 0,C 180,E1 20991,E2 20991} C_VEL
LIN {X 0,Y 440.798,Z 783.037,A -85,B 0,C 180,E1 20989.064,E2 20989.064} C_VEL
LIN {X 0,Y 440.875,Z 781.188,A -85,B 0,C 180,E1 20987.011,E2 20987.011} C_VEL
LIN {X 0,Y 441.069,Z 777.593,A -85,B 0,C 180,E1 20985.049,E2 20985.049} C_VEL
LIN {X 0,Y 441.396,Z 772.559,A -85,B 0,C 180,E1 20983.225,E2 20983.225} C_VEL
LIN {X 0,Y 441.901,Z 765.348,A -85,B 0,C 180,E1 20981.353,E2 20981.353} C_VEL
LIN {X 0,Y 442.492,Z 757.324,A -85,B 0,C 180,E1 20979.757,E2 20979.757} C_VEL
LIN {X 0,Y 443.255,Z 747.11,A -85,B 0,C 180,E1 20978.17,E2 20978.17} C_VEL
LIN {X 0,Y 444.058,Z 735.8,A -85,B 0,C 180,E1 20976.792,E2 20976.792} C_VEL
LIN {X 0,Y 444.865,Z 723.521,A -85,B 0,C 180,E1 20975.61,E2 20975.61} C_VEL
LIN {X 0,Y 445.664,Z 709.325,A -85,B 0,C 180,E1 20974.568,E2 20974.568} C_VEL
LIN {X 0,Y 446.291,Z 694.943,A -85,B 0,C 180,E1 20973.789,E2 20973.789} C_VEL
LIN {X 0,Y 446.748,Z 679.523,A -85,B 0,C 180,E1 20973.216,E2 20973.216} C_VEL
LIN {X 0,Y 447.05,Z 658.68,A -85,B 0,C 180,E1 20972.79,E2 20972.79} C_VEL
LIN {X 0,Y 448.039,Z 574.052,A -85,B 0,C 180,E1 20971.362,E2 20971.362} C_VEL
LIN {X 0,Y 444.694,Z 555.082,A -85,B 0,C 180,E1 20970.837,E2 20970.837} C_VEL
LIN {X 0,Y 446.344,Z 525.878,A -85,B 0,C 180,E1 20966.918,E2 20966.918} C_VEL
LIN {X 0,Y 448.267,Z 497.811,A -85,B 0,C 180,E1 20963.082,E2 20963.082} C_VEL
LIN {X 0,Y 449.729,Z 478.485,A -85,B 0,C 180,E1 20960.401,E2 20960.401} C_VEL
LIN {X 0,Y 444.689,Z 459.877,A -85,B 0,C 180,E1 20957.27,E2 20957.27} C_VEL
LIN {X 0,Y 441.165,Z 447.975,A -85,B 0,C 180,E1 20955.127,E2 20955.127} C_VEL
LIN {X 0,Y 441.18,Z 447.842,A -85,B 0,C 180,E1 20951.501,E2 20951.501} C_VEL
LIN {X 0,Y 441.155,Z 447.819,A -85,B 0,C 180,E1 20947.759,E2 20947.759} C_VEL
LIN {X 0,Y 441.13,Z 447.845,A -85,B 0,C 180,E1 20944.058,E2 20944.058} C_VEL
LIN {X 0,Y 441.118,Z 447.848,A -85,B 0,C 180,E1 20940.387,E2 20940.387} C_VEL
LIN {X 0,Y 441.133,Z 447.846,A -85,B 0,C 180,E1 20936.735,E2 20936.735} C_VEL
LIN {X 0,Y 441.169,Z 447.832,A -85,B 0,C 180,E1 20933.087,E2 20933.087} C_VEL
LIN {X 0,Y 441.161,Z 447.842,A -85,B 0,C 180,E1 20929.399,E2 20929.399} C_VEL
LIN {X 0,Y 441.135,Z 447.842,A -85,B 0,C 180,E1 20925.725,E2 20925.725} C_VEL
LIN {X 0,Y 441.128,Z 447.832,A -85,B 0,C 180,E1 20921.974,E2 20921.974} C_VEL
LIN {X 0,Y 441.138,Z 447.845,A -85,B 0,C 180,E1 20918.227,E2 20918.227} C_VEL
LIN {X 0,Y 441.171,Z 447.819,A -85,B 0,C 180,E1 20914.644,E2 20914.644} C_VEL
LIN {X 0,Y 441.198,Z 447.843,A -85,B 0,C 180,E1 20910.806,E2 20910.806} C_VEL
LIN {X 0,Y 441.166,Z 447.823,A -85,B 0,C 180,E1 20907.101,E2 20907.101} C_VEL
LIN {X 0,Y 441.143,Z 447.839,A -85,B 0,C 180,E1 20903.51,E2 20903.51} C_VEL
LIN {X 0,Y 441.145,Z 447.835,A -85,B 0,C 180,E1 20899.738,E2 20899.738} C_VEL
LIN {X 0,Y 441.165,Z 447.831,A -85,B 0,C 180,E1 20896.052,E2 20896.052} C_VEL
LIN {X 0,Y 441.195,Z 447.837,A -85,B 0,C 180,E1 20892.376,E2 20892.376} C_VEL
LIN {X 0,Y 441.186,Z 447.814,A -85,B 0,C 180,E1 20888.603,E2 20888.603} C_VEL
LIN {X 0,Y 441.163,Z 447.84,A -85,B 0,C 180,E1 20884.941,E2 20884.941} C_VEL
LIN {X 0,Y 441.154,Z 447.827,A -85,B 0,C 180,E1 20881.169,E2 20881.169} C_VEL
LIN {X 0,Y 441.161,Z 447.838,A -85,B 0,C 180,E1 20877.402,E2 20877.402} C_VEL
LIN {X 0,Y 441.186,Z 447.828,A -85,B 0,C 180,E1 20873.755,E2 20873.755} C_VEL
LIN {X 0,Y 441.198,Z 447.837,A -85,B 0,C 180,E1 20869.951,E2 20869.951} C_VEL
LIN {X 0,Y 441.198,Z 447.826,A -85,B 0,C 180,E1 20866.101,E2 20866.101} C_VEL
LIN {X 0,Y 441.188,Z 447.84,A -85,B 0,C 180,E1 20862.321,E2 20862.321} C_VEL
LIN {X 0,Y 441.172,Z 447.828,A -85,B 0,C 180,E1 20858.6,E2 20858.6} C_VEL
LIN {X 0,Y 441.172,Z 447.841,A -85,B 0,C 180,E1 20854.781,E2 20854.781} C_VEL
LIN {X 0,Y 441.178,Z 447.84,A -85,B 0,C 180,E1 20850.988,E2 20850.988} C_VEL
LIN {X 0,Y 441.193,Z 447.837,A -85,B 0,C 180,E1 20847.224,E2 20847.224} C_VEL
LIN {X 0,Y 441.196,Z 447.836,A -85,B 0,C 180,E1 20843.415,E2 20843.415} C_VEL
LIN {X 0,Y 441.196,Z 447.839,A -85,B 0,C 180,E1 20839.593,E2 20839.593} C_VEL
LIN {X 0,Y 441.195,Z 447.841,A -85,B 0,C 180,E1 20835.737,E2 20835.737} C_VEL
LIN {X 0,Y 441.19,Z 447.837,A -85,B 0,C 180,E1 20831.956,E2 20831.956} C_VEL
LIN {X 0,Y 441.23,Z 448.106,A -85,B 0,C 180,E1 20829.425,E2 20829.425} C_VEL
LIN {X 0,Y 449.046,Z 470.12,A -85,B 0,C 180,E1 20826.397,E2 20826.397} C_VEL
LIN {X 0,Y 454.138,Z 485.498,A -85,B 0,C 180,E1 20824.46,E2 20824.46} C_VEL
LIN {X 0,Y 450.639,Z 529.524,A -85,B 0,C 180,E1 20820.43,E2 20820.43} C_VEL
LIN {X 0,Y 449.922,Z 540.505,A -85,B 0,C 180,E1 20819.456,E2 20819.456} C_VEL
LIN {X 0,Y 452.283,Z 562.105,A -85,B 0,C 180,E1 20818.949,E2 20818.949} C_VEL
LIN {X 0,Y 449.945,Z 741.748,A -85,B 0,C 180,E1 20816.059,E2 20816.059} C_VEL
LIN {X 0,Y 449.185,Z 760.538,A -85,B 0,C 180,E1 20815.531,E2 20815.531} C_VEL
LIN {X 0,Y 448.188,Z 778.422,A -85,B 0,C 180,E1 20814.798,E2 20814.798} C_VEL
LIN {X 0,Y 447.06,Z 796.002,A -85,B 0,C 180,E1 20813.832,E2 20813.832} C_VEL
LIN {X 0,Y 445.809,Z 813.26,A -85,B 0,C 180,E1 20812.622,E2 20812.622} C_VEL
LIN {X 0,Y 444.577,Z 829.263,A -85,B 0,C 180,E1 20811.229,E2 20811.229} C_VEL
LIN {X 0,Y 443.408,Z 844.29,A -85,B 0,C 180,E1 20809.633,E2 20809.633} C_VEL
LIN {X 0,Y 442.391,Z 857.825,A -85,B 0,C 180,E1 20807.901,E2 20807.901} C_VEL
LIN {X 0,Y 441.58,Z 869.991,A -85,B 0,C 180,E1 20806.036,E2 20806.036} C_VEL
LIN {X 0,Y 440.932,Z 881.31,A -85,B 0,C 180,E1 20803.944,E2 20803.944} C_VEL
LIN {X 0,Y 440.546,Z 890.823,A -85,B 0,C 180,E1 20801.787,E2 20801.787} C_VEL
LIN {X 0,Y 440.347,Z 898.728,A -85,B 0,C 180,E1 20799.541,E2 20799.541} C_VEL
LIN {X 0,Y 440.313,Z 905.098,A -85,B 0,C 180,E1 20797.175,E2 20797.175} C_VEL
LIN {X 0,Y 440.365,Z 909.559,A -85,B 0,C 180,E1 20794.819,E2 20794.819} C_VEL
LIN {X 0,Y 440.43,Z 912.218,A -85,B 0,C 180,E1 20792.472,E2 20792.472} C_VEL
LIN {X 0,Y 440.47,Z 913.142,A -85,B 0,C 180,E1 20790.13,E2 20790.13} C_VEL
LIN {X 0,Y 440.449,Z 912.348,A -85,B 0,C 180,E1 20787.789,E2 20787.789} C_VEL
LIN {X 0,Y 440.39,Z 909.83,A -85,B 0,C 180,E1 20785.442,E2 20785.442} C_VEL
LIN {X 0,Y 440.333,Z 905.535,A -85,B 0,C 180,E1 20783.088,E2 20783.088} C_VEL
LIN {X 0,Y 440.347,Z 899.741,A -85,B 0,C 180,E1 20780.855,E2 20780.855} C_VEL
LIN {X 0,Y 440.512,Z 892.143,A -85,B 0,C 180,E1 20778.611,E2 20778.611} C_VEL
LIN {X 0,Y 440.841,Z 883.137,A -85,B 0,C 180,E1 20776.49,E2 20776.49} C_VEL
LIN {X 0,Y 441.427,Z 872.078,A -85,B 0,C 180,E1 20774.363,E2 20774.363} C_VEL
LIN {X 0,Y 442.252,Z 859.464,A -85,B 0,C 180,E1 20772.365,E2 20772.365} C_VEL
LIN {X 0,Y 443.308,Z 845.166,A -85,B 0,C 180,E1 20770.5,E2 20770.5} C_VEL
LIN {X 0,Y 444.463,Z 830.443,A -85,B 0,C 180,E1 20768.904,E2 20768.904} C_VEL
LIN {X 0,Y 445.671,Z 814.891,A -85,B 0,C 180,E1 20767.511,E2 20767.511} C_VEL
LIN {X 0,Y 446.889,Z 798.745,A -85,B 0,C 180,E1 20766.331,E2 20766.331} C_VEL
LIN {X 0,Y 448.057,Z 781.623,A -85,B 0,C 180,E1 20765.336,E2 20765.336} C_VEL
LIN {X 0,Y 449.117,Z 763.553,A -85,B 0,C 180,E1 20764.541,E2 20764.541} C_VEL
LIN {X 0,Y 449.967,Z 744.689,A -85,B 0,C 180,E1 20763.965,E2 20763.965} C_VEL
LIN {X 0,Y 450.465,Z 718.42,A -85,B 0,C 180,E1 20763.49,E2 20763.49} C_VEL
LIN {X 0,Y 452.41,Z 559.139,A -85,B 0,C 180,E1 20760.91,E2 20760.91} C_VEL
LIN {X 0,Y 450.242,Z 540.374,A -85,B 0,C 180,E1 20760.417,E2 20760.417} C_VEL
LIN {X 0,Y 453.898,Z 496.922,A -85,B 0,C 180,E1 20756.374,E2 20756.374} C_VEL
LIN {X 0,Y 454.795,Z 485.741,A -85,B 0,C 180,E1 20755.291,E2 20755.291} C_VEL
LIN {X 0,Y 448.755,Z 467.701,A -85,B 0,C 180,E1 20752.8,E2 20752.8} C_VEL
LIN {X 0,Y 442.358,Z 451.129,A -85,B 0,C 180,E1 20750.219,E2 20750.219} C_VEL
LIN {X 0,Y 441.209,Z 448.007,A -85,B 0,C 180,E1 20749.642,E2 20749.642} C_VEL
LIN {X 0,Y 441.192,Z 447.842,A -85,B 0,C 180,E1 20745.914,E2 20745.914} C_VEL
LIN {X 0,Y 441.194,Z 447.833,A -85,B 0,C 180,E1 20742.13,E2 20742.13} C_VEL
LIN {X 0,Y 441.19,Z 447.834,A -85,B 0,C 180,E1 20738.36,E2 20738.36} C_VEL
LIN {X 0,Y 441.192,Z 447.838,A -85,B 0,C 180,E1 20734.511,E2 20734.511} C_VEL
LIN {X 0,Y 441.199,Z 447.837,A -85,B 0,C 180,E1 20730.657,E2 20730.657} C_VEL
LIN {X 0,Y 441.186,Z 447.839,A -85,B 0,C 180,E1 20726.953,E2 20726.953} C_VEL
LIN {X 0,Y 441.184,Z 447.832,A -85,B 0,C 180,E1 20723.224,E2 20723.224} C_VEL
LIN {X 0,Y 441.191,Z 447.827,A -85,B 0,C 180,E1 20719.459,E2 20719.459} C_VEL
LIN {X 0,Y 441.195,Z 447.831,A -85,B 0,C 180,E1 20715.645,E2 20715.645} C_VEL
LIN {X 0,Y 441.192,Z 447.84,A -85,B 0,C 180,E1 20711.901,E2 20711.901} C_VEL
LIN {X 0,Y 441.197,Z 447.834,A -85,B 0,C 180,E1 20708.077,E2 20708.077} C_VEL
LIN {X 0,Y 441.186,Z 447.825,A -85,B 0,C 180,E1 20704.289,E2 20704.289} C_VEL
LIN {X 0,Y 441.178,Z 447.829,A -85,B 0,C 180,E1 20700.519,E2 20700.519} C_VEL
LIN {X 0,Y 441.182,Z 447.84,A -85,B 0,C 180,E1 20696.752,E2 20696.752} C_VEL
LIN {X 0,Y 441.2,Z 447.841,A -85,B 0,C 180,E1 20692.97,E2 20692.97} C_VEL
LIN {X 0,Y 441.193,Z 447.834,A -85,B 0,C 180,E1 20689.158,E2 20689.158} C_VEL
LIN {X 0,Y 441.195,Z 447.83,A -85,B 0,C 180,E1 20685.395,E2 20685.395} C_VEL
LIN {X 0,Y 441.192,Z 447.833,A -85,B 0,C 180,E1 20681.638,E2 20681.638} C_VEL
LIN {X 0,Y 441.18,Z 447.84,A -85,B 0,C 180,E1 20677.9,E2 20677.9} C_VEL
LIN {X 0,Y 441.179,Z 447.844,A -85,B 0,C 180,E1 20674.061,E2 20674.061} C_VEL
LIN {X 0,Y 441.185,Z 447.836,A -85,B 0,C 180,E1 20670.243,E2 20670.243} C_VEL
LIN {X 0,Y 441.194,Z 447.842,A -85,B 0,C 180,E1 20666.429,E2 20666.429} C_VEL
LIN {X 0,Y 441.242,Z 448.267,A -85,B 0,C 180,E1 20665.925,E2 20665.925} C_VEL
LIN {X 0,Y 446.222,Z 463.416,A -85,B 0,C 180,E1 20662.91,E2 20662.91} C_VEL
LIN {X 0,Y 450.502,Z 478.875,A -85,B 0,C 180,E1 20660.102,E2 20660.102} C_VEL
LIN {X 0,Y 450.916,Z 481.62,A -85,B 0,C 180,E1 20659.648,E2 20659.648} C_VEL
LIN {X 0,Y 448.483,Z 509.531,A -85,B 0,C 180,E1 20655.696,E2 20655.696} C_VEL
LIN {X 0,Y 446.415,Z 537.82,A -85,B 0,C 180,E1 20651.768,E2 20651.768} C_VEL
LIN {X 0,Y 445.348,Z 555.128,A -85,B 0,C 180,E1 20649.437,E2 20649.437} C_VEL
LIN {X 0,Y 449.209,Z 576.623,A -85,B 0,C 180,E1 20648.784,E2 20648.784} C_VEL
LIN {X 0,Y 447.557,Z 675.852,A -85,B 0,C 180,E1 20647.043,E2 20647.043} C_VEL
LIN {X 0,Y 447.133,Z 692.173,A -85,B 0,C 180,E1 20646.499,E2 20646.499} C_VEL
LIN {X 0,Y 446.501,Z 706.629,A -85,B 0,C 180,E1 20645.765,E2 20645.765} C_VEL
LIN {X 0,Y 445.694,Z 720.527,A -85,B 0,C 180,E1 20644.807,E2 20644.807} C_VEL
LIN {X 0,Y 445.542,Z 722.708,A -85,B 0,C 180,E1 20644.628,E2 20644.628} C_VEL
LIN {X 0,Y 444.169,Z 729.213,A -85,B 0,C 180,E1 20644.108,E2 20644.108} C_VEL
LIN {X 0,Y 438.739,Z 741.452,A -85,B 0,C 180,E1 20643.055,E2 20643.055} C_VEL
LIN {X 0,Y 436.309,Z 747.917,A -85,B 0,C 180,E1 20642.323,E2 20642.323} C_VEL
LIN {X 0,Y 435.916,Z 750.174,A -85,B 0,C 180,E1 20642.009,E2 20642.009} C_VEL
LIN {X 0,Y 435.025,Z 760.095,A -85,B 0,C 180,E1 20640.374,E2 20640.374} C_VEL
LIN {X 0,Y 434.222,Z 768.93,A -85,B 0,C 180,E1 20638.466,E2 20638.466} C_VEL
LIN {X 0,Y 433.625,Z 775.524,A -85,B 0,C 180,E1 20636.535,E2 20636.535} C_VEL
LIN {X 0,Y 433.229,Z 780.293,A -85,B 0,C 180,E1 20634.546,E2 20634.546} C_VEL
LIN {X 0,Y 432.99,Z 783.374,A -85,B 0,C 180,E1 20632.396,E2 20632.396} C_VEL
LIN {X 0,Y 432.889,Z 784.425,A -85,B 0,C 180,E1 20630.271,E2 20630.271} C_VEL
LIN {X 0,Y 432.903,Z 783.751,A -85,B 0,C 180,E1 20628.307,E2 20628.307} C_VEL
LIN {X 0,Y 433.039,Z 781.108,A -85,B 0,C 180,E1 20626.152,E2 20626.152} C_VEL
LIN {X 0,Y 433.305,Z 776.758,A -85,B 0,C 180,E1 20624.158,E2 20624.158} C_VEL
LIN {X 0,Y 433.749,Z 770.717,A -85,B 0,C 180,E1 20622.244,E2 20622.244} C_VEL
LIN {X 0,Y 434.385,Z 762.537,A -85,B 0,C 180,E1 20620.343,E2 20620.343} C_VEL
LIN {X 0,Y 435.102,Z 753.428,A -85,B 0,C 180,E1 20618.723,E2 20618.723} C_VEL
LIN {X 0,Y 435.931,Z 742.956,A -85,B 0,C 180,E1 20617.247,E2 20617.247} C_VEL
LIN {X 0,Y 436.847,Z 730.211,A -85,B 0,C 180,E1 20615.846,E2 20615.846} C_VEL
LIN {X 0,Y 437.664,Z 717.77,A -85,B 0,C 180,E1 20614.783,E2 20614.783} C_VEL
LIN {X 0,Y 438.425,Z 703.711,A -85,B 0,C 180,E1 20613.86,E2 20613.86} C_VEL
LIN {X 0,Y 439.015,Z 688.299,A -85,B 0,C 180,E1 20613.141,E2 20613.141} C_VEL
LIN {X 0,Y 439.374,Z 673.1,A -85,B 0,C 180,E1 20612.686,E2 20612.686} C_VEL
LIN {X 0,Y 440.612,Z 575.027,A -85,B 0,C 180,E1 20610.983,E2 20610.983} C_VEL
LIN {X 0,Y 437.079,Z 555.045,A -85,B 0,C 180,E1 20610.426,E2 20610.426} C_VEL
LIN {X 0,Y 438.831,Z 525.935,A -85,B 0,C 180,E1 20606.473,E2 20606.473} C_VEL
LIN {X 0,Y 440.874,Z 497.821,A -85,B 0,C 180,E1 20602.572,E2 20602.572} C_VEL
LIN {X 0,Y 442.086,Z 480.357,A -85,B 0,C 180,E1 20600.102,E2 20600.102} C_VEL
LIN {X 0,Y 437.168,Z 462.213,A -85,B 0,C 180,E1 20596.988,E2 20596.988} C_VEL
LIN {X 0,Y 433.208,Z 448.972,A -85,B 0,C 180,E1 20594.573,E2 20594.573} C_VEL
LIN {X 0,Y 433.194,Z 448.831,A -85,B 0,C 180,E1 20590.867,E2 20590.867} C_VEL
LIN {X 0,Y 433.215,Z 448.799,A -85,B 0,C 180,E1 20587.186,E2 20587.186} C_VEL
LIN {X 0,Y 433.233,Z 448.835,A -85,B 0,C 180,E1 20583.401,E2 20583.401} C_VEL
LIN {X 0,Y 433.21,Z 448.837,A -85,B 0,C 180,E1 20579.638,E2 20579.638} C_VEL
LIN {X 0,Y 433.186,Z 448.835,A -85,B 0,C 180,E1 20575.959,E2 20575.959} C_VEL
LIN {X 0,Y 433.183,Z 448.829,A -85,B 0,C 180,E1 20572.29,E2 20572.29} C_VEL
LIN {X 0,Y 433.206,Z 448.822,A -85,B 0,C 180,E1 20568.692,E2 20568.692} C_VEL
LIN {X 0,Y 433.234,Z 448.834,A -85,B 0,C 180,E1 20564.928,E2 20564.928} C_VEL
LIN {X 0,Y 433.238,Z 448.812,A -85,B 0,C 180,E1 20561.129,E2 20561.129} C_VEL
LIN {X 0,Y 433.209,Z 448.835,A -85,B 0,C 180,E1 20557.442,E2 20557.442} C_VEL
LIN {X 0,Y 433.194,Z 448.811,A -85,B 0,C 180,E1 20553.798,E2 20553.798} C_VEL
LIN {X 0,Y 433.204,Z 448.833,A -85,B 0,C 180,E1 20550.057,E2 20550.057} C_VEL
LIN {X 0,Y 433.232,Z 448.803,A -85,B 0,C 180,E1 20546.431,E2 20546.431} C_VEL
LIN {X 0,Y 433.26,Z 448.831,A -85,B 0,C 180,E1 20542.615,E2 20542.615} C_VEL
LIN {X 0,Y 433.238,Z 448.809,A -85,B 0,C 180,E1 20538.851,E2 20538.851} C_VEL
LIN {X 0,Y 433.217,Z 448.823,A -85,B 0,C 180,E1 20535.118,E2 20535.118} C_VEL
LIN {X 0,Y 433.21,Z 448.828,A -85,B 0,C 180,E1 20531.449,E2 20531.449} C_VEL
LIN {X 0,Y 433.217,Z 448.812,A -85,B 0,C 180,E1 20527.693,E2 20527.693} C_VEL
LIN {X 0,Y 433.242,Z 448.827,A -85,B 0,C 180,E1 20523.97,E2 20523.97} C_VEL
LIN {X 0,Y 433.263,Z 448.8,A -85,B 0,C 180,E1 20520.132,E2 20520.132} C_VEL
LIN {X 0,Y 433.255,Z 448.832,A -85,B 0,C 180,E1 20516.295,E2 20516.295} C_VEL
LIN {X 0,Y 433.237,Z 448.81,A -85,B 0,C 180,E1 20512.574,E2 20512.574} C_VEL
LIN {X 0,Y 433.226,Z 448.83,A -85,B 0,C 180,E1 20508.822,E2 20508.822} C_VEL
LIN {X 0,Y 433.224,Z 448.812,A -85,B 0,C 180,E1 20505.02,E2 20505.02} C_VEL
LIN {X 0,Y 433.24,Z 448.829,A -85,B 0,C 180,E1 20501.289,E2 20501.289} C_VEL
LIN {X 0,Y 433.259,Z 448.82,A -85,B 0,C 180,E1 20497.475,E2 20497.475} C_VEL
LIN {X 0,Y 433.258,Z 448.815,A -85,B 0,C 180,E1 20493.699,E2 20493.699} C_VEL
LIN {X 0,Y 433.263,Z 448.827,A -85,B 0,C 180,E1 20489.929,E2 20489.929} C_VEL
LIN {X 0,Y 433.254,Z 448.833,A -85,B 0,C 180,E1 20486.049,E2 20486.049} C_VEL
LIN {X 0,Y 433.243,Z 448.832,A -85,B 0,C 180,E1 20482.296,E2 20482.296} C_VEL
LIN {X 0,Y 433.243,Z 448.832,A -85,B 0,C 180,E1 20478.521,E2 20478.521} C_VEL
LIN {X 0,Y 433.247,Z 448.824,A -85,B 0,C 180,E1 20474.699,E2 20474.699} C_VEL
LIN {X 0,Y 433.262,Z 448.831,A -85,B 0,C 180,E1 20470.95,E2 20470.95} C_VEL
LIN {X 0,Y 433.297,Z 449.141,A -85,B 0,C 180,E1 20470.029,E2 20470.029} C_VEL
LIN {X 0,Y 441.256,Z 471.42,A -85,B 0,C 180,E1 20466.882,E2 20466.882} C_VEL
LIN {X 0,Y 446.755,Z 488.134,A -85,B 0,C 180,E1 20464.729,E2 20464.729} C_VEL
LIN {X 0,Y 443.084,Z 531.777,A -85,B 0,C 180,E1 20460.663,E2 20460.663} C_VEL
LIN {X 0,Y 442.498,Z 541.014,A -85,B 0,C 180,E1 20459.852,E2 20459.852} C_VEL
LIN {X 0,Y 444.896,Z 563.055,A -85,B 0,C 180,E1 20459.332,E2 20459.332} C_VEL
LIN {X 0,Y 442.438,Z 741.128,A -85,B 0,C 180,E1 20456.423,E2 20456.423} C_VEL
LIN {X 0,Y 441.637,Z 759.924,A -85,B 0,C 180,E1 20455.886,E2 20455.886} C_VEL
LIN {X 0,Y 440.6,Z 777.675,A -85,B 0,C 180,E1 20455.146,E2 20455.146} C_VEL
LIN {X 0,Y 439.392,Z 795.525,A -85,B 0,C 180,E1 20454.148,E2 20454.148} C_VEL
LIN {X 0,Y 438.062,Z 812.902,A -85,B 0,C 180,E1 20452.902,E2 20452.902} C_VEL
LIN {X 0,Y 436.763,Z 828.818,A -85,B 0,C 180,E1 20451.487,E2 20451.487} C_VEL
LIN {X 0,Y 435.545,Z 843.81,A -85,B 0,C 180,E1 20449.862,E2 20449.862} C_VEL
LIN {X 0,Y 434.446,Z 857.788,A -85,B 0,C 180,E1 20448.032,E2 20448.032} C_VEL
LIN {X 0,Y 433.581,Z 870.202,A -85,B 0,C 180,E1 20446.065,E2 20446.065} C_VEL
LIN {X 0,Y 432.92,Z 881.457,A -85,B 0,C 180,E1 20443.898,E2 20443.898} C_VEL
LIN {X 0,Y 432.536,Z 891.082,A -85,B 0,C 180,E1 20441.602,E2 20441.602} C_VEL
LIN {X 0,Y 432.37,Z 898.677,A -85,B 0,C 180,E1 20439.316,E2 20439.316} C_VEL
LIN {X 0,Y 432.365,Z 904.462,A -85,B 0,C 180,E1 20437.04,E2 20437.04} C_VEL
LIN {X 0,Y 432.434,Z 908.578,A -85,B 0,C 180,E1 20434.767,E2 20434.767} C_VEL
LIN {X 0,Y 432.513,Z 911.149,A -85,B 0,C 180,E1 20432.385,E2 20432.385} C_VEL
LIN {X 0,Y 432.558,Z 911.991,A -85,B 0,C 180,E1 20430,E2 20430} C_VEL
LIN {X 0,Y 432.52,Z 911.099,A -85,B 0,C 180,E1 20427.615,E2 20427.615} C_VEL
LIN {X 0,Y 432.445,Z 908.459,A -85,B 0,C 180,E1 20425.216,E2 20425.216} C_VEL
LIN {X 0,Y 432.374,Z 903.94,A -85,B 0,C 180,E1 20422.772,E2 20422.772} C_VEL
LIN {X 0,Y 432.387,Z 897.741,A -85,B 0,C 180,E1 20420.416,E2 20420.416} C_VEL
LIN {X 0,Y 432.578,Z 889.879,A -85,B 0,C 180,E1 20418.129,E2 20418.129} C_VEL
LIN {X 0,Y 432.968,Z 880.305,A -85,B 0,C 180,E1 20415.909,E2 20415.909} C_VEL
LIN {X 0,Y 433.626,Z 869.172,A -85,B 0,C 180,E1 20413.8,E2 20413.8} C_VEL
LIN {X 0,Y 434.477,Z 857.022,A -85,B 0,C 180,E1 20411.885,E2 20411.885} C_VEL
LIN {X 0,Y 435.582,Z 843.187,A -85,B 0,C 180,E1 20410.07,E2 20410.07} C_VEL
LIN {X 0,Y 436.83,Z 828.146,A -85,B 0,C 180,E1 20408.435,E2 20408.435} C_VEL
LIN {X 0,Y 438.221,Z 811.569,A -85,B 0,C 180,E1 20406.961,E2 20406.961} C_VEL
LIN {X 0,Y 439.542,Z 794.77,A -85,B 0,C 180,E1 20405.758,E2 20405.758} C_VEL
LIN {X 0,Y 440.797,Z 776.961,A -85,B 0,C 180,E1 20404.758,E2 20404.758} C_VEL
LIN {X 0,Y 441.888,Z 758.841,A -85,B 0,C 180,E1 20404.003,E2 20404.003} C_VEL
LIN {X 0,Y 442.716,Z 739.989,A -85,B 0,C 180,E1 20403.469,E2 20403.469} C_VEL
LIN {X 0,Y 445.18,Z 560.07,A -85,B 0,C 180,E1 20400.481,E2 20400.481} C_VEL
LIN {X 0,Y 442.951,Z 540.499,A -85,B 0,C 180,E1 20399.949,E2 20399.949} C_VEL
LIN {X 0,Y 446.897,Z 497.236,A -85,B 0,C 180,E1 20395.836,E2 20395.836} C_VEL
LIN {X 0,Y 447.74,Z 489.016,A -85,B 0,C 180,E1 20395.04,E2 20395.04} C_VEL
LIN {X 0,Y 441.768,Z 471.034,A -85,B 0,C 180,E1 20392.495,E2 20392.495} C_VEL
LIN {X 0,Y 435.815,Z 455.525,A -85,B 0,C 180,E1 20390.02,E2 20390.02} C_VEL
LIN {X 0,Y 433.283,Z 449.018,A -85,B 0,C 180,E1 20388.853,E2 20388.853} C_VEL
LIN {X 0,Y 433.253,Z 448.823,A -85,B 0,C 180,E1 20385.075,E2 20385.075} C_VEL
LIN {X 0,Y 433.25,Z 448.829,A -85,B 0,C 180,E1 20381.206,E2 20381.206} C_VEL
LIN {X 0,Y 433.246,Z 448.831,A -85,B 0,C 180,E1 20377.37,E2 20377.37} C_VEL
LIN {X 0,Y 433.248,Z 448.827,A -85,B 0,C 180,E1 20373.475,E2 20373.475} C_VEL
LIN {X 0,Y 433.256,Z 448.826,A -85,B 0,C 180,E1 20369.595,E2 20369.595} C_VEL
LIN {X 0,Y 433.255,Z 448.83,A -85,B 0,C 180,E1 20365.713,E2 20365.713} C_VEL
LIN {X 0,Y 433.254,Z 448.829,A -85,B 0,C 180,E1 20361.917,E2 20361.917} C_VEL
LIN {X 0,Y 433.254,Z 448.822,A -85,B 0,C 180,E1 20358.046,E2 20358.046} C_VEL
LIN {X 0,Y 433.258,Z 448.809,A -85,B 0,C 180,E1 20354.244,E2 20354.244} C_VEL
LIN {X 0,Y 433.251,Z 448.818,A -85,B 0,C 180,E1 20350.37,E2 20350.37} C_VEL
LIN {X 0,Y 433.241,Z 448.828,A -85,B 0,C 180,E1 20346.626,E2 20346.626} C_VEL
LIN {X 0,Y 433.243,Z 448.832,A -85,B 0,C 180,E1 20342.778,E2 20342.778} C_VEL
LIN {X 0,Y 433.25,Z 448.817,A -85,B 0,C 180,E1 20338.942,E2 20338.942} C_VEL
LIN {X 0,Y 433.252,Z 448.815,A -85,B 0,C 180,E1 20335.101,E2 20335.101} C_VEL
LIN {X 0,Y 433.254,Z 448.822,A -85,B 0,C 180,E1 20331.372,E2 20331.372} C_VEL
LIN {X 0,Y 433.257,Z 448.828,A -85,B 0,C 180,E1 20327.606,E2 20327.606} C_VEL
LIN {X 0,Y 433.252,Z 448.828,A -85,B 0,C 180,E1 20323.785,E2 20323.785} C_VEL
LIN {X 0,Y 433.243,Z 448.829,A -85,B 0,C 180,E1 20319.933,E2 20319.933} C_VEL
LIN {X 0,Y 433.241,Z 448.824,A -85,B 0,C 180,E1 20316.179,E2 20316.179} C_VEL
LIN {X 0,Y 433.248,Z 448.824,A -85,B 0,C 180,E1 20312.362,E2 20312.362} C_VEL
LIN {X 0,Y 433.257,Z 448.829,A -85,B 0,C 180,E1 20308.563,E2 20308.563} C_VEL
LIN {X 0,Y 433.299,Z 449.118,A -85,B 0,C 180,E1 20306.724,E2 20306.724} C_VEL
LIN {X 0,Y 438.288,Z 464.189,A -85,B 0,C 180,E1 20303.62,E2 20303.62} C_VEL
LIN {X 0,Y 442.547,Z 479.145,A -85,B 0,C 180,E1 20300.8,E2 20300.8} C_VEL
LIN {X 0,Y 443.638,Z 483.972,A -85,B 0,C 180,E1 20299.95,E2 20299.95} C_VEL
LIN {X 0,Y 441.048,Z 511.832,A -85,B 0,C 180,E1 20295.942,E2 20295.942} C_VEL
LIN {X 0,Y 438.853,Z 539.986,A -85,B 0,C 180,E1 20291.975,E2 20291.975} C_VEL
LIN {X 0,Y 437.863,Z 554.607,A -85,B 0,C 180,E1 20289.958,E2 20289.958} C_VEL
LIN {X 0,Y 440.572,Z 568.887,A -85,B 0,C 180,E1 20289.473,E2 20289.473} C_VEL
LIN {X 0,Y 441.996,Z 578.328,A -85,B 0,C 180,E1 20289.21,E2 20289.21} C_VEL
LIN {X 0,Y 440.247,Z 676.403,A -85,B 0,C 180,E1 20287.457,E2 20287.457} C_VEL
LIN {X 0,Y 439.791,Z 692.674,A -85,B 0,C 180,E1 20286.906,E2 20286.906} C_VEL
LIN {X 0,Y 439.167,Z 706.302,A -85,B 0,C 180,E1 20286.214,E2 20286.214} C_VEL
LIN {X 0,Y 438.31,Z 720.389,A -85,B 0,C 180,E1 20285.248,E2 20285.248} C_VEL
LIN {X 0,Y 437.311,Z 733.422,A -85,B 0,C 180,E1 20284.067,E2 20284.067} C_VEL
LIN {X 0,Y 436.381,Z 744.945,A -85,B 0,C 180,E1 20282.734,E2 20282.734} C_VEL
LIN {X 0,Y 435.916,Z 750.174,A -85,B 0,C 180,E1 20282.009,E2 20282.009} C_VEL
LIN {X 0,Y 434.514,Z 755.348,A -85,B 0,C 180,E1 20281.264,E2 20281.264} C_VEL
LIN {X 0,Y 429.468,Z 764.203,A -85,B 0,C 180,E1 20279.889,E2 20279.889} C_VEL
LIN {X 0,Y 426.907,Z 768.968,A -85,B 0,C 180,E1 20278.943,E2 20278.943} C_VEL
LIN {X 0,Y 426.352,Z 771.055,A -85,B 0,C 180,E1 20278.424,E2 20278.424} C_VEL
LIN {X 0,Y 425.744,Z 777.272,A -85,B 0,C 180,E1 20276.501,E2 20276.501} C_VEL
LIN {X 0,Y 425.333,Z 781.714,A -85,B 0,C 180,E1 20274.529,E2 20274.529} C_VEL
LIN {X 0,Y 425.085,Z 784.616,A -85,B 0,C 180,E1 20272.398,E2 20272.398} C_VEL
LIN {X 0,Y 424.974,Z 785.61,A -85,B 0,C 180,E1 20270.156,E2 20270.156} C_VEL
LIN {X 0,Y 424.994,Z 784.742,A -85,B 0,C 180,E1 20268.092,E2 20268.092} C_VEL
LIN {X 0,Y 425.149,Z 782.066,A -85,B 0,C 180,E1 20265.971,E2 20265.971} C_VEL
LIN {X 0,Y 425.464,Z 777.416,A -85,B 0,C 180,E1 20263.869,E2 20263.869} C_VEL
LIN {X 0,Y 425.912,Z 771.7,A -85,B 0,C 180,E1 20262.06,E2 20262.06} C_VEL
LIN {X 0,Y 426.598,Z 763.488,A -85,B 0,C 180,E1 20260.124,E2 20260.124} C_VEL
LIN {X 0,Y 427.365,Z 754.345,A -85,B 0,C 180,E1 20258.476,E2 20258.476} C_VEL
LIN {X 0,Y 428.246,Z 743.848,A -85,B 0,C 180,E1 20256.973,E2 20256.973} C_VEL
LIN {X 0,Y 429.217,Z 731.073,A -85,B 0,C 180,E1 20255.547,E2 20255.547} C_VEL
LIN {X 0,Y 430.078,Z 718.612,A -85,B 0,C 180,E1 20254.467,E2 20254.467} C_VEL
LIN {X 0,Y 430.88,Z 704.5,A -85,B 0,C 180,E1 20253.525,E2 20253.525} C_VEL
LIN {X 0,Y 431.499,Z 689.098,A -85,B 0,C 180,E1 20252.794,E2 20252.794} C_VEL
LIN {X 0,Y 431.879,Z 673.897,A -85,B 0,C 180,E1 20252.328,E2 20252.328} C_VEL
LIN {X 0,Y 433.188,Z 576.043,A -85,B 0,C 180,E1 20250.599,E2 20250.599} C_VEL
LIN {X 0,Y 429.48,Z 555.012,A -85,B 0,C 180,E1 20250,E2 20250} C_VEL
LIN {X 0,Y 430.127,Z 543.127,A -85,B 0,C 180,E1 20248.401,E2 20248.401} C_VEL
LIN {X 0,Y 432.169,Z 514.664,A -85,B 0,C 180,E1 20244.423,E2 20244.423} C_VEL
LIN {X 0,Y 434.439,Z 486.677,A -85,B 0,C 180,E1 20240.461,E2 20240.461} C_VEL
LIN {X 0,Y 434.63,Z 483.019,A -85,B 0,C 180,E1 20239.931,E2 20239.931} C_VEL
LIN {X 0,Y 429.829,Z 465.187,A -85,B 0,C 180,E1 20236.822,E2 20236.822} C_VEL
LIN {X 0,Y 425.289,Z 449.926,A -85,B 0,C 180,E1 20233.964,E2 20233.964} C_VEL
LIN {X 0,Y 425.254,Z 449.822,A -85,B 0,C 180,E1 20230.21,E2 20230.21} C_VEL
LIN {X 0,Y 425.242,Z 449.789,A -85,B 0,C 180,E1 20226.439,E2 20226.439} C_VEL
LIN {X 0,Y 425.25,Z 449.822,A -85,B 0,C 180,E1 20222.71,E2 20222.71} C_VEL
LIN {X 0,Y 425.272,Z 449.819,A -85,B 0,C 180,E1 20219.009,E2 20219.009} C_VEL
LIN {X 0,Y 425.289,Z 449.822,A -85,B 0,C 180,E1 20215.159,E2 20215.159} C_VEL
LIN {X 0,Y 425.296,Z 449.818,A -85,B 0,C 180,E1 20211.291,E2 20211.291} C_VEL
LIN {X 0,Y 425.265,Z 449.807,A -85,B 0,C 180,E1 20207.563,E2 20207.563} C_VEL
LIN {X 0,Y 425.252,Z 449.823,A -85,B 0,C 180,E1 20203.917,E2 20203.917} C_VEL
LIN {X 0,Y 425.254,Z 449.815,A -85,B 0,C 180,E1 20200.108,E2 20200.108} C_VEL
LIN {X 0,Y 425.277,Z 449.815,A -85,B 0,C 180,E1 20196.479,E2 20196.479} C_VEL
LIN {X 0,Y 425.303,Z 449.806,A -85,B 0,C 180,E1 20192.686,E2 20192.686} C_VEL
LIN {X 0,Y 425.304,Z 449.815,A -85,B 0,C 180,E1 20188.966,E2 20188.966} C_VEL
LIN {X 0,Y 425.281,Z 449.797,A -85,B 0,C 180,E1 20185.155,E2 20185.155} C_VEL
LIN {X 0,Y 425.267,Z 449.822,A -85,B 0,C 180,E1 20181.517,E2 20181.517} C_VEL
LIN {X 0,Y 425.266,Z 449.79,A -85,B 0,C 180,E1 20177.656,E2 20177.656} C_VEL
LIN {X 0,Y 425.279,Z 449.819,A -85,B 0,C 180,E1 20173.833,E2 20173.833} C_VEL
LIN {X 0,Y 425.304,Z 449.797,A -85,B 0,C 180,E1 20170.156,E2 20170.156} C_VEL
LIN {X 0,Y 425.321,Z 449.807,A -85,B 0,C 180,E1 20166.344,E2 20166.344} C_VEL
LIN {X 0,Y 425.314,Z 449.807,A -85,B 0,C 180,E1 20162.426,E2 20162.426} C_VEL
LIN {X 0,Y 425.297,Z 449.801,A -85,B 0,C 180,E1 20158.653,E2 20158.653} C_VEL
LIN {X 0,Y 425.288,Z 449.821,A -85,B 0,C 180,E1 20154.875,E2 20154.875} C_VEL
LIN {X 0,Y 425.282,Z 449.802,A -85,B 0,C 180,E1 20151.074,E2 20151.074} C_VEL
LIN {X 0,Y 425.29,Z 449.817,A -85,B 0,C 180,E1 20147.233,E2 20147.233} C_VEL
LIN {X 0,Y 425.307,Z 449.811,A -85,B 0,C 180,E1 20143.474,E2 20143.474} C_VEL
LIN {X 0,Y 425.319,Z 449.805,A -85,B 0,C 180,E1 20139.64,E2 20139.64} C_VEL
LIN {X 0,Y 425.321,Z 449.819,A -85,B 0,C 180,E1 20135.801,E2 20135.801} C_VEL
LIN {X 0,Y 425.321,Z 449.808,A -85,B 0,C 180,E1 20131.955,E2 20131.955} C_VEL
LIN {X 0,Y 425.308,Z 449.808,A -85,B 0,C 180,E1 20128.224,E2 20128.224} C_VEL
LIN {X 0,Y 425.3,Z 449.812,A -85,B 0,C 180,E1 20124.433,E2 20124.433} C_VEL
LIN {X 0,Y 425.298,Z 449.811,A -85,B 0,C 180,E1 20120.598,E2 20120.598} C_VEL
LIN {X 0,Y 425.309,Z 449.816,A -85,B 0,C 180,E1 20116.785,E2 20116.785} C_VEL
LIN {X 0,Y 425.317,Z 449.819,A -85,B 0,C 180,E1 20112.981,E2 20112.981} C_VEL
LIN {X 0,Y 425.35,Z 450.084,A -85,B 0,C 180,E1 20110.672,E2 20110.672} C_VEL
LIN {X 0,Y 432.883,Z 471.127,A -85,B 0,C 180,E1 20107.604,E2 20107.604} C_VEL
LIN {X 0,Y 439.397,Z 490.496,A -85,B 0,C 180,E1 20105.031,E2 20105.031} C_VEL
LIN {X 0,Y 435.453,Z 534.808,A -85,B 0,C 180,E1 20100.823,E2 20100.823} C_VEL
LIN {X 0,Y 435.061,Z 541.185,A -85,B 0,C 180,E1 20100.268,E2 20100.268} C_VEL
LIN {X 0,Y 437.519,Z 563.998,A -85,B 0,C 180,E1 20099.724,E2 20099.724} C_VEL
LIN {X 0,Y 434.948,Z 740.506,A -85,B 0,C 180,E1 20096.799,E2 20096.799} C_VEL
LIN {X 0,Y 434.117,Z 759.146,A -85,B 0,C 180,E1 20096.259,E2 20096.259} C_VEL
LIN {X 0,Y 433.023,Z 777.063,A -85,B 0,C 180,E1 20095.501,E2 20095.501} C_VEL
LIN {X 0,Y 431.755,Z 794.817,A -85,B 0,C 180,E1 20094.49,E2 20094.49} C_VEL
LIN {X 0,Y 430.328,Z 812.544,A -85,B 0,C 180,E1 20093.193,E2 20093.193} C_VEL
LIN {X 0,Y 428.96,Z 828.36,A -85,B 0,C 180,E1 20091.754,E2 20091.754} C_VEL
LIN {X 0,Y 427.686,Z 843.268,A -85,B 0,C 180,E1 20090.1,E2 20090.1} C_VEL
LIN {X 0,Y 426.572,Z 856.687,A -85,B 0,C 180,E1 20088.306,E2 20088.306} C_VEL
LIN {X 0,Y 425.633,Z 869.542,A -85,B 0,C 180,E1 20086.233,E2 20086.233} C_VEL
LIN {X 0,Y 424.95,Z 880.729,A -85,B 0,C 180,E1 20084.025,E2 20084.025} C_VEL
LIN {X 0,Y 424.575,Z 889.808,A -85,B 0,C 180,E1 20081.823,E2 20081.823} C_VEL
LIN {X 0,Y 424.402,Z 897.44,A -85,B 0,C 180,E1 20079.493,E2 20079.493} C_VEL
LIN {X 0,Y 424.411,Z 903.255,A -85,B 0,C 180,E1 20077.173,E2 20077.173} C_VEL
LIN {X 0,Y 424.497,Z 907.38,A -85,B 0,C 180,E1 20074.864,E2 20074.864} C_VEL
LIN {X 0,Y 424.591,Z 909.977,A -85,B 0,C 180,E1 20072.43,E2 20072.43} C_VEL
LIN {X 0,Y 424.643,Z 910.824,A -85,B 0,C 180,E1 20070,E2 20070} C_VEL
LIN {X 0,Y 424.598,Z 909.928,A -85,B 0,C 180,E1 20067.571,E2 20067.571} C_VEL
LIN {X 0,Y 424.506,Z 907.208,A -85,B 0,C 180,E1 20065.077,E2 20065.077} C_VEL
LIN {X 0,Y 424.418,Z 902.785,A -85,B 0,C 180,E1 20062.66,E2 20062.66} C_VEL
LIN {X 0,Y 424.422,Z 896.504,A -85,B 0,C 180,E1 20060.235,E2 20060.235} C_VEL
LIN {X 0,Y 424.618,Z 888.616,A -85,B 0,C 180,E1 20057.903,E2 20057.903} C_VEL
LIN {X 0,Y 425.015,Z 879.318,A -85,B 0,C 180,E1 20055.699,E2 20055.699} C_VEL
LIN {X 0,Y 425.734,Z 867.88,A -85,B 0,C 180,E1 20053.491,E2 20053.491} C_VEL
LIN {X 0,Y 426.645,Z 855.794,A -85,B 0,C 180,E1 20051.556,E2 20051.556} C_VEL
LIN {X 0,Y 427.851,Z 841.671,A -85,B 0,C 180,E1 20049.68,E2 20049.68} C_VEL
LIN {X 0,Y 429.222,Z 826.091,A -85,B 0,C 180,E1 20047.973,E2 20047.973} C_VEL
LIN {X 0,Y 430.667,Z 809.941,A -85,B 0,C 180,E1 20046.53,E2 20046.53} C_VEL
LIN {X 0,Y 432.071,Z 793.041,A -85,B 0,C 180,E1 20045.311,E2 20045.311} C_VEL
LIN {X 0,Y 433.374,Z 775.728,A -85,B 0,C 180,E1 20044.331,E2 20044.331} C_VEL
LIN {X 0,Y 434.522,Z 757.526,A -85,B 0,C 180,E1 20043.565,E2 20043.565} C_VEL
LIN {X 0,Y 435.401,Z 738.459,A -85,B 0,C 180,E1 20043.025,E2 20043.025} C_VEL
LIN {X 0,Y 437.994,Z 561.023,A -85,B 0,C 180,E1 20040.035,E2 20040.035} C_VEL
LIN {X 0,Y 435.692,Z 540.65,A -85,B 0,C 180,E1 20039.468,E2 20039.468} C_VEL
LIN {X 0,Y 439.996,Z 496.967,A -85,B 0,C 180,E1 20035.224,E2 20035.224} C_VEL
LIN {X 0,Y 440.567,Z 491.886,A -85,B 0,C 180,E1 20034.72,E2 20034.72} C_VEL
LIN {X 0,Y 434.98,Z 474.886,A -85,B 0,C 180,E1 20032.254,E2 20032.254} C_VEL
LIN {X 0,Y 429.085,Z 459.511,A -85,B 0,C 180,E1 20029.742,E2 20029.742} C_VEL
LIN {X 0,Y 425.341,Z 450.005,A -85,B 0,C 180,E1 20027.997,E2 20027.997} C_VEL
LIN {X 0,Y 425.315,Z 449.813,A -85,B 0,C 180,E1 20024.192,E2 20024.192} C_VEL
LIN {X 0,Y 425.315,Z 449.818,A -85,B 0,C 180,E1 20020.277,E2 20020.277} C_VEL
LIN {X 0,Y 425.314,Z 449.812,A -85,B 0,C 180,E1 20016.487,E2 20016.487} C_VEL
LIN {X 0,Y 425.316,Z 449.807,A -85,B 0,C 180,E1 20012.571,E2 20012.571} C_VEL
LIN {X 0,Y 425.318,Z 449.806,A -85,B 0,C 180,E1 20008.734,E2 20008.734} C_VEL
LIN {X 0,Y 425.31,Z 449.81,A -85,B 0,C 180,E1 20004.846,E2 20004.846} C_VEL
LIN {X 0,Y 425.307,Z 449.816,A -85,B 0,C 180,E1 20001.043,E2 20001.043} C_VEL
LIN {X 0,Y 425.31,Z 449.822,A -85,B 0,C 180,E1 19997.23,E2 19997.23} C_VEL
LIN {X 0,Y 425.316,Z 449.806,A -85,B 0,C 180,E1 19993.458,E2 19993.458} C_VEL
LIN {X 0,Y 425.314,Z 449.801,A -85,B 0,C 180,E1 19989.608,E2 19989.608} C_VEL
LIN {X 0,Y 425.316,Z 449.811,A -85,B 0,C 180,E1 19985.802,E2 19985.802} C_VEL
LIN {X 0,Y 425.316,Z 449.817,A -85,B 0,C 180,E1 19981.886,E2 19981.886} C_VEL
LIN {X 0,Y 425.31,Z 449.815,A -85,B 0,C 180,E1 19978.114,E2 19978.114} C_VEL
LIN {X 0,Y 425.302,Z 449.807,A -85,B 0,C 180,E1 19974.333,E2 19974.333} C_VEL
LIN {X 0,Y 425.302,Z 449.804,A -85,B 0,C 180,E1 19970.528,E2 19970.528} C_VEL
LIN {X 0,Y 425.309,Z 449.806,A -85,B 0,C 180,E1 19966.68,E2 19966.68} C_VEL
LIN {X 0,Y 425.316,Z 449.809,A -85,B 0,C 180,E1 19962.911,E2 19962.911} C_VEL
LIN {X 0,Y 425.318,Z 449.809,A -85,B 0,C 180,E1 19959.063,E2 19959.063} C_VEL
LIN {X 0,Y 425.319,Z 449.809,A -85,B 0,C 180,E1 19955.152,E2 19955.152} C_VEL
LIN {X 0,Y 425.324,Z 449.819,A -85,B 0,C 180,E1 19951.265,E2 19951.265} C_VEL
LIN {X 0,Y 425.329,Z 449.987,A -85,B 0,C 180,E1 19947.589,E2 19947.589} C_VEL
LIN {X 0,Y 430.192,Z 464.408,A -85,B 0,C 180,E1 19944.475,E2 19944.475} C_VEL
LIN {X 0,Y 434.54,Z 479.156,A -85,B 0,C 180,E1 19941.591,E2 19941.591} C_VEL
LIN {X 0,Y 436.301,Z 487.122,A -85,B 0,C 180,E1 19940.148,E2 19940.148} C_VEL
LIN {X 0,Y 433.547,Z 515.471,A -85,B 0,C 180,E1 19936.017,E2 19936.017} C_VEL
LIN {X 0,Y 431.189,Z 543.619,A -85,B 0,C 180,E1 19931.989,E2 19931.989} C_VEL
LIN {X 0,Y 430.45,Z 554.628,A -85,B 0,C 180,E1 19930.467,E2 19930.467} C_VEL
LIN {X 0,Y 433.827,Z 572.293,A -85,B 0,C 180,E1 19929.86,E2 19929.86} C_VEL
LIN {X 0,Y 434.816,Z 579.627,A -85,B 0,C 180,E1 19929.656,E2 19929.656} C_VEL
LIN {X 0,Y 432.964,Z 677.003,A -85,B 0,C 180,E1 19927.884,E2 19927.884} C_VEL
LIN {X 0,Y 432.478,Z 693.266,A -85,B 0,C 180,E1 19927.326,E2 19927.326} C_VEL
LIN {X 0,Y 431.763,Z 707.852,A -85,B 0,C 180,E1 19926.568,E2 19926.568} C_VEL
LIN {X 0,Y 430.886,Z 721.322,A -85,B 0,C 180,E1 19925.622,E2 19925.622} C_VEL
LIN {X 0,Y 429.821,Z 734.362,A -85,B 0,C 180,E1 19924.421,E2 19924.421} C_VEL
LIN {X 0,Y 428.819,Z 745.894,A -85,B 0,C 180,E1 19923.066,E2 19923.066} C_VEL
LIN {X 0,Y 427.76,Z 756.889,A -85,B 0,C 180,E1 19921.416,E2 19921.416} C_VEL
LIN {X 0,Y 426.907,Z 765.437,A -85,B 0,C 180,E1 19919.77,E2 19919.77} C_VEL
LIN {X 0,Y 426.352,Z 771.055,A -85,B 0,C 180,E1 19918.424,E2 19918.424} C_VEL
LIN {X 0,Y 425.051,Z 774.511,A -85,B 0,C 180,E1 19917.5,E2 19917.5} C_VEL
LIN {X 0,Y 420.221,Z 780.174,A -85,B 0,C 180,E1 19915.805,E2 19915.805} C_VEL
LIN {X 0,Y 417.74,Z 782.997,A -85,B 0,C 180,E1 19914.617,E2 19914.617} C_VEL
LIN {X 0,Y 417.377,Z 783.848,A -85,B 0,C 180,E1 19914.099,E2 19914.099} C_VEL
LIN {X 0,Y 417.132,Z 786.293,A -85,B 0,C 180,E1 19911.81,E2 19911.81} C_VEL
LIN {X 0,Y 417.05,Z 786.703,A -85,B 0,C 180,E1 19909.611,E2 19909.611} C_VEL
LIN {X 0,Y 417.111,Z 785.313,A -85,B 0,C 180,E1 19907.435,E2 19907.435} C_VEL
LIN {X 0,Y 417.321,Z 782.052,A -85,B 0,C 180,E1 19905.281,E2 19905.281} C_VEL
LIN {X 0,Y 417.686,Z 777.23,A -85,B 0,C 180,E1 19903.285,E2 19903.285} C_VEL
LIN {X 0,Y 418.265,Z 770.539,A -85,B 0,C 180,E1 19901.304,E2 19901.304} C_VEL
LIN {X 0,Y 418.991,Z 762.274,A -85,B 0,C 180,E1 19899.477,E2 19899.477} C_VEL
LIN {X 0,Y 419.865,Z 752.566,A -85,B 0,C 180,E1 19897.801,E2 19897.801} C_VEL
LIN {X 0,Y 420.89,Z 740.737,A -85,B 0,C 180,E1 19896.205,E2 19896.205} C_VEL
LIN {X 0,Y 421.891,Z 727.797,A -85,B 0,C 180,E1 19894.854,E2 19894.854} C_VEL
LIN {X 0,Y 422.79,Z 714.757,A -85,B 0,C 180,E1 19893.797,E2 19893.797} C_VEL
LIN {X 0,Y 423.607,Z 699.635,A -85,B 0,C 180,E1 19892.878,E2 19892.878} C_VEL
LIN {X 0,Y 424.173,Z 683.927,A -85,B 0,C 180,E1 19892.225,E2 19892.225} C_VEL
LIN {X 0,Y 424.489,Z 667.884,A -85,B 0,C 180,E1 19891.824,E2 19891.824} C_VEL
LIN {X 0,Y 425.792,Z 577.165,A -85,B 0,C 180,E1 19890.208,E2 19890.208} C_VEL
LIN {X 0,Y 421.884,Z 554.956,A -85,B 0,C 180,E1 19889.562,E2 19889.562} C_VEL
LIN {X 0,Y 422.077,Z 549.918,A -85,B 0,C 180,E1 19888.914,E2 19888.914} C_VEL
LIN {X 0,Y 424.277,Z 520.362,A -85,B 0,C 180,E1 19884.726,E2 19884.726} C_VEL
LIN {X 0,Y 426.563,Z 493.12,A -85,B 0,C 180,E1 19880.828,E2 19880.828} C_VEL
LIN {X 0,Y 427.183,Z 485.693,A -85,B 0,C 180,E1 19879.753,E2 19879.753} C_VEL
LIN {X 0,Y 422.395,Z 467.802,A -85,B 0,C 180,E1 19876.586,E2 19876.586} C_VEL
LIN {X 0,Y 417.367,Z 450.936,A -85,B 0,C 180,E1 19873.372,E2 19873.372} C_VEL
LIN {X 0,Y 417.361,Z 450.812,A -85,B 0,C 180,E1 19869.507,E2 19869.507} C_VEL
LIN {X 0,Y 417.34,Z 450.779,A -85,B 0,C 180,E1 19865.664,E2 19865.664} C_VEL
LIN {X 0,Y 417.322,Z 450.804,A -85,B 0,C 180,E1 19861.836,E2 19861.836} C_VEL
LIN {X 0,Y 417.302,Z 450.806,A -85,B 0,C 180,E1 19858.189,E2 19858.189} C_VEL
LIN {X 0,Y 417.305,Z 450.81,A -85,B 0,C 180,E1 19854.316,E2 19854.316} C_VEL
LIN {X 0,Y 417.316,Z 450.814,A -85,B 0,C 180,E1 19850.488,E2 19850.488} C_VEL
LIN {X 0,Y 417.336,Z 450.8,A -85,B 0,C 180,E1 19846.747,E2 19846.747} C_VEL
LIN {X 0,Y 417.361,Z 450.799,A -85,B 0,C 180,E1 19843.056,E2 19843.056} C_VEL
LIN {X 0,Y 417.349,Z 450.804,A -85,B 0,C 180,E1 19839.233,E2 19839.233} C_VEL
LIN {X 0,Y 417.329,Z 450.796,A -85,B 0,C 180,E1 19835.437,E2 19835.437} C_VEL
LIN {X 0,Y 417.322,Z 450.807,A -85,B 0,C 180,E1 19831.649,E2 19831.649} C_VEL
LIN {X 0,Y 417.323,Z 450.8,A -85,B 0,C 180,E1 19827.853,E2 19827.853} C_VEL
LIN {X 0,Y 417.333,Z 450.804,A -85,B 0,C 180,E1 19824.035,E2 19824.035} C_VEL
LIN {X 0,Y 417.36,Z 450.8,A -85,B 0,C 180,E1 19820.327,E2 19820.327} C_VEL
LIN {X 0,Y 417.372,Z 450.782,A -85,B 0,C 180,E1 19816.421,E2 19816.421} C_VEL
LIN {X 0,Y 417.374,Z 450.807,A -85,B 0,C 180,E1 19812.592,E2 19812.592} C_VEL
LIN {X 0,Y 417.363,Z 450.777,A -85,B 0,C 180,E1 19808.681,E2 19808.681} C_VEL
LIN {X 0,Y 417.347,Z 450.807,A -85,B 0,C 180,E1 19804.948,E2 19804.948} C_VEL
LIN {X 0,Y 417.339,Z 450.788,A -85,B 0,C 180,E1 19801.098,E2 19801.098} C_VEL
LIN {X 0,Y 417.342,Z 450.805,A -85,B 0,C 180,E1 19797.254,E2 19797.254} C_VEL
LIN {X 0,Y 417.347,Z 450.796,A -85,B 0,C 180,E1 19793.397,E2 19793.397} C_VEL
LIN {X 0,Y 417.367,Z 450.805,A -85,B 0,C 180,E1 19789.65,E2 19789.65} C_VEL
LIN {X 0,Y 417.382,Z 450.787,A -85,B 0,C 180,E1 19785.715,E2 19785.715} C_VEL
LIN {X 0,Y 417.384,Z 450.807,A -85,B 0,C 180,E1 19781.855,E2 19781.855} C_VEL
LIN {X 0,Y 417.384,Z 450.79,A -85,B 0,C 180,E1 19777.908,E2 19777.908} C_VEL
LIN {X 0,Y 417.377,Z 450.796,A -85,B 0,C 180,E1 19773.999,E2 19773.999} C_VEL
LIN {X 0,Y 417.378,Z 450.809,A -85,B 0,C 180,E1 19770.114,E2 19770.114} C_VEL
LIN {X 0,Y 417.369,Z 450.809,A -85,B 0,C 180,E1 19766.231,E2 19766.231} C_VEL
LIN {X 0,Y 417.364,Z 450.81,A -85,B 0,C 180,E1 19762.346,E2 19762.346} C_VEL
LIN {X 0,Y 417.364,Z 450.809,A -85,B 0,C 180,E1 19758.426,E2 19758.426} C_VEL
LIN {X 0,Y 417.367,Z 450.802,A -85,B 0,C 180,E1 19754.582,E2 19754.582} C_VEL
LIN {X 0,Y 417.41,Z 451.04,A -85,B 0,C 180,E1 19751.341,E2 19751.341} C_VEL
LIN {X 0,Y 424.763,Z 471.497,A -85,B 0,C 180,E1 19748.249,E2 19748.249} C_VEL
LIN {X 0,Y 432.012,Z 493.133,A -85,B 0,C 180,E1 19745.312,E2 19745.312} C_VEL
LIN {X 0,Y 427.78,Z 538.269,A -85,B 0,C 180,E1 19740.945,E2 19740.945} C_VEL
LIN {X 0,Y 427.663,Z 541.647,A -85,B 0,C 180,E1 19740.686,E2 19740.686} C_VEL
LIN {X 0,Y 430.137,Z 564.894,A -85,B 0,C 180,E1 19740.122,E2 19740.122} C_VEL
LIN {X 0,Y 427.451,Z 740.04,A -85,B 0,C 180,E1 19737.176,E2 19737.176} C_VEL
LIN {X 0,Y 426.579,Z 758.723,A -85,B 0,C 180,E1 19736.626,E2 19736.626} C_VEL
LIN {X 0,Y 425.422,Z 776.9,A -85,B 0,C 180,E1 19735.84,E2 19735.84} C_VEL
LIN {X 0,Y 424.095,Z 794.579,A -85,B 0,C 180,E1 19734.812,E2 19734.812} C_VEL
LIN {X 0,Y 422.677,Z 811.341,A -85,B 0,C 180,E1 19733.564,E2 19733.564} C_VEL
LIN {X 0,Y 421.255,Z 826.932,A -85,B 0,C 180,E1 19732.128,E2 19732.128} C_VEL
LIN {X 0,Y 419.943,Z 841.569,A -85,B 0,C 180,E1 19730.487,E2 19730.487} C_VEL
LIN {X 0,Y 418.75,Z 855.101,A -85,B 0,C 180,E1 19728.66,E2 19728.66} C_VEL
LIN {X 0,Y 417.801,Z 867.243,A -85,B 0,C 180,E1 19726.689,E2 19726.689} C_VEL
LIN {X 0,Y 417.086,Z 878.027,A -85,B 0,C 180,E1 19724.579,E2 19724.579} C_VEL
LIN {X 0,Y 416.656,Z 887.431,A -85,B 0,C 180,E1 19722.332,E2 19722.332} C_VEL
LIN {X 0,Y 416.451,Z 895.373,A -85,B 0,C 180,E1 19719.955,E2 19719.955} C_VEL
LIN {X 0,Y 416.448,Z 901.771,A -85,B 0,C 180,E1 19717.441,E2 19717.441} C_VEL
LIN {X 0,Y 416.561,Z 906.192,A -85,B 0,C 180,E1 19714.957,E2 19714.957} C_VEL
LIN {X 0,Y 416.668,Z 908.804,A -85,B 0,C 180,E1 19712.476,E2 19712.476} C_VEL
LIN {X 0,Y 416.729,Z 909.656,A -85,B 0,C 180,E1 19710,E2 19710} C_VEL
LIN {X 0,Y 416.676,Z 908.757,A -85,B 0,C 180,E1 19707.525,E2 19707.525} C_VEL
LIN {X 0,Y 416.572,Z 906.108,A -85,B 0,C 180,E1 19705.043,E2 19705.043} C_VEL
LIN {X 0,Y 416.459,Z 901.653,A -85,B 0,C 180,E1 19702.548,E2 19702.548} C_VEL
LIN {X 0,Y 416.455,Z 895.299,A -85,B 0,C 180,E1 19700.046,E2 19700.046} C_VEL
LIN {X 0,Y 416.663,Z 887.123,A -85,B 0,C 180,E1 19697.599,E2 19697.599} C_VEL
LIN {X 0,Y 417.12,Z 877.393,A -85,B 0,C 180,E1 19695.281,E2 19695.281} C_VEL
LIN {X 0,Y 417.86,Z 866.533,A -85,B 0,C 180,E1 19693.161,E2 19693.161} C_VEL
LIN {X 0,Y 418.877,Z 853.97,A -85,B 0,C 180,E1 19691.129,E2 19691.129} C_VEL
LIN {X 0,Y 420.179,Z 839.81,A -85,B 0,C 180,E1 19689.234,E2 19689.234} C_VEL
LIN {X 0,Y 421.598,Z 824.664,A -85,B 0,C 180,E1 19687.553,E2 19687.553} C_VEL
LIN {X 0,Y 423.142,Z 808.565,A -85,B 0,C 180,E1 19686.094,E2 19686.094} C_VEL
LIN {X 0,Y 424.641,Z 791.491,A -85,B 0,C 180,E1 19684.849,E2 19684.849} C_VEL
LIN {X 0,Y 426.04,Z 773.985,A -85,B 0,C 180,E1 19683.857,E2 19683.857} C_VEL
LIN {X 0,Y 427.257,Z 755.477,A -85,B 0,C 180,E1 19683.082,E2 19683.082} C_VEL
LIN {X 0,Y 428.12,Z 736.412,A -85,B 0,C 180,E1 19682.558,E2 19682.558} C_VEL
LIN {X 0,Y 430.847,Z 562.046,A -85,B 0,C 180,E1 19679.575,E2 19679.575} C_VEL
LIN {X 0,Y 428.459,Z 541.139,A -85,B 0,C 180,E1 19678.993,E2 19678.993} C_VEL
LIN {X 0,Y 433.075,Z 497.525,A -85,B 0,C 180,E1 19674.666,E2 19674.666} C_VEL
LIN {X 0,Y 433.284,Z 494.284,A -85,B 0,C 180,E1 19674.32,E2 19674.32} C_VEL
LIN {X 0,Y 427.683,Z 477.23,A -85,B 0,C 180,E1 19671.768,E2 19671.768} C_VEL
LIN {X 0,Y 421.711,Z 461.597,A -85,B 0,C 180,E1 19669.127,E2 19669.127} C_VEL
LIN {X 0,Y 417.426,Z 451.14,A -85,B 0,C 180,E1 19667.135,E2 19667.135} C_VEL
LIN {X 0,Y 417.371,Z 450.807,A -85,B 0,C 180,E1 19665.749,E2 19665.749} C_VEL
LIN {X 0,Y 417.375,Z 450.799,A -85,B 0,C 180,E1 19661.839,E2 19661.839} C_VEL
LIN {X 0,Y 417.379,Z 450.804,A -85,B 0,C 180,E1 19657.988,E2 19657.988} C_VEL
LIN {X 0,Y 417.38,Z 450.81,A -85,B 0,C 180,E1 19654.018,E2 19654.018} C_VEL
LIN {X 0,Y 417.378,Z 450.809,A -85,B 0,C 180,E1 19650.044,E2 19650.044} C_VEL
LIN {X 0,Y 417.376,Z 450.807,A -85,B 0,C 180,E1 19646.154,E2 19646.154} C_VEL
LIN {X 0,Y 417.379,Z 450.803,A -85,B 0,C 180,E1 19642.241,E2 19642.241} C_VEL
LIN {X 0,Y 417.378,Z 450.798,A -85,B 0,C 180,E1 19638.289,E2 19638.289} C_VEL
LIN {X 0,Y 417.377,Z 450.786,A -85,B 0,C 180,E1 19634.426,E2 19634.426} C_VEL
LIN {X 0,Y 417.369,Z 450.796,A -85,B 0,C 180,E1 19630.49,E2 19630.49} C_VEL
LIN {X 0,Y 417.364,Z 450.806,A -85,B 0,C 180,E1 19626.603,E2 19626.603} C_VEL
LIN {X 0,Y 417.365,Z 450.809,A -85,B 0,C 180,E1 19622.746,E2 19622.746} C_VEL
LIN {X 0,Y 417.372,Z 450.794,A -85,B 0,C 180,E1 19618.902,E2 19618.902} C_VEL
LIN {X 0,Y 417.373,Z 450.791,A -85,B 0,C 180,E1 19615.052,E2 19615.052} C_VEL
LIN {X 0,Y 417.377,Z 450.795,A -85,B 0,C 180,E1 19611.181,E2 19611.181} C_VEL
LIN {X 0,Y 417.377,Z 450.8,A -85,B 0,C 180,E1 19607.268,E2 19607.268} C_VEL
LIN {X 0,Y 417.38,Z 450.803,A -85,B 0,C 180,E1 19603.38,E2 19603.38} C_VEL
LIN {X 0,Y 417.38,Z 450.801,A -85,B 0,C 180,E1 19599.498,E2 19599.498} C_VEL
LIN {X 0,Y 417.371,Z 450.797,A -85,B 0,C 180,E1 19595.666,E2 19595.666} C_VEL
LIN {X 0,Y 417.364,Z 450.805,A -85,B 0,C 180,E1 19591.836,E2 19591.836} C_VEL
LIN {X 0,Y 417.415,Z 451.08,A -85,B 0,C 180,E1 19588.425,E2 19588.425} C_VEL
LIN {X 0,Y 422.396,Z 465.432,A -85,B 0,C 180,E1 19585.216,E2 19585.216} C_VEL
LIN {X 0,Y 426.702,Z 479.842,A -85,B 0,C 180,E1 19582.296,E2 19582.296} C_VEL
LIN {X 0,Y 429.072,Z 489.539,A -85,B 0,C 180,E1 19580.473,E2 19580.473} C_VEL
LIN {X 0,Y 426.145,Z 517.896,A -85,B 0,C 180,E1 19576.274,E2 19576.274} C_VEL
LIN {X 0,Y 423.633,Z 546.131,A -85,B 0,C 180,E1 19572.174,E2 19572.174} C_VEL
LIN {X 0,Y 423.05,Z 554.393,A -85,B 0,C 180,E1 19571.015,E2 19571.015} C_VEL
LIN {X 0,Y 424.445,Z 561.819,A -85,B 0,C 180,E1 19570.716,E2 19570.716} C_VEL
LIN {X 0,Y 427.681,Z 580.259,A -85,B 0,C 180,E1 19570.131,E2 19570.131} C_VEL
LIN {X 0,Y 425.703,Z 677.634,A -85,B 0,C 180,E1 19568.325,E2 19568.325} C_VEL
LIN {X 0,Y 425.19,Z 693.837,A -85,B 0,C 180,E1 19567.761,E2 19567.761} C_VEL
LIN {X 0,Y 424.447,Z 708.247,A -85,B 0,C 180,E1 19567.005,E2 19567.005} C_VEL
LIN {X 0,Y 423.48,Z 722.271,A -85,B 0,C 180,E1 19566.008,E2 19566.008} C_VEL
LIN {X 0,Y 422.324,Z 735.551,A -85,B 0,C 180,E1 19564.761,E2 19564.761} C_VEL
LIN {X 0,Y 421.272,Z 746.843,A -85,B 0,C 180,E1 19563.41,E2 19563.41} C_VEL
LIN {X 0,Y 420.108,Z 758.107,A -85,B 0,C 180,E1 19561.689,E2 19561.689} C_VEL
LIN {X 0,Y 419.135,Z 767.105,A -85,B 0,C 180,E1 19559.906,E2 19559.906} C_VEL
LIN {X 0,Y 418.376,Z 774.213,A -85,B 0,C 180,E1 19558.086,E2 19558.086} C_VEL
LIN {X 0,Y 417.739,Z 780.202,A -85,B 0,C 180,E1 19555.977,E2 19555.977} C_VEL
LIN {X 0,Y 417.377,Z 783.848,A -85,B 0,C 180,E1 19554.099,E2 19554.099} C_VEL
LIN {X 0,Y 416.24,Z 785.363,A -85,B 0,C 180,E1 19553.061,E2 19553.061} C_VEL
LIN {X 0,Y 411.855,Z 787.381,A -85,B 0,C 180,E1 19551.243,E2 19551.243} C_VEL
LIN {X 0,Y 409.402,Z 787.899,A -85,B 0,C 180,E1 19549.885,E2 19549.885} C_VEL
LIN {X 0,Y 409.137,Z 787.808,A -85,B 0,C 180,E1 19549.341,E2 19549.341} C_VEL
LIN {X 0,Y 409.209,Z 786.208,A -85,B 0,C 180,E1 19547.181,E2 19547.181} C_VEL
LIN {X 0,Y 409.453,Z 782.806,A -85,B 0,C 180,E1 19545.001,E2 19545.001} C_VEL
LIN {X 0,Y 409.901,Z 777.37,A -85,B 0,C 180,E1 19542.825,E2 19542.825} C_VEL
LIN {X 0,Y 410.494,Z 770.884,A -85,B 0,C 180,E1 19540.952,E2 19540.952} C_VEL
LIN {X 0,Y 411.292,Z 762.443,A -85,B 0,C 180,E1 19539.092,E2 19539.092} C_VEL
LIN {X 0,Y 412.235,Z 752.466,A -85,B 0,C 180,E1 19537.386,E2 19537.386} C_VEL
LIN {X 0,Y 413.228,Z 741.591,A -85,B 0,C 180,E1 19535.909,E2 19535.909} C_VEL
LIN {X 0,Y 414.258,Z 728.936,A -85,B 0,C 180,E1 19534.563,E2 19534.563} C_VEL
LIN {X 0,Y 415.234,Z 715.484,A -85,B 0,C 180,E1 19533.451,E2 19533.451} C_VEL
LIN {X 0,Y 416.061,Z 700.922,A -85,B 0,C 180,E1 19532.548,E2 19532.548} C_VEL
LIN {X 0,Y 416.658,Z 685.585,A -85,B 0,C 180,E1 19531.884,E2 19531.884} C_VEL
LIN {X 0,Y 417.008,Z 669.662,A -85,B 0,C 180,E1 19531.462,E2 19531.462} C_VEL
LIN {X 0,Y 418.412,Z 578.257,A -85,B 0,C 180,E1 19529.803,E2 19529.803} C_VEL
LIN {X 0,Y 414.281,Z 554.714,A -85,B 0,C 180,E1 19529.101,E2 19529.101} C_VEL
LIN {X 0,Y 415.17,Z 541.35,A -85,B 0,C 180,E1 19527.239,E2 19527.239} C_VEL
LIN {X 0,Y 417.502,Z 512.752,A -85,B 0,C 180,E1 19523.122,E2 19523.122} C_VEL
LIN {X 0,Y 419.718,Z 488.384,A -85,B 0,C 180,E1 19519.569,E2 19519.569} C_VEL
LIN {X 0,Y 415.198,Z 471.237,A -85,B 0,C 180,E1 19516.491,E2 19516.491} C_VEL
LIN {X 0,Y 410.176,Z 454.402,A -85,B 0,C 180,E1 19513.283,E2 19513.283} C_VEL
LIN {X 0,Y 409.391,Z 451.923,A -85,B 0,C 180,E1 19512.737,E2 19512.737} C_VEL
LIN {X 0,Y 409.385,Z 451.801,A -85,B 0,C 180,E1 19508.959,E2 19508.959} C_VEL
LIN {X 0,Y 409.408,Z 451.772,A -85,B 0,C 180,E1 19505.3,E2 19505.3} C_VEL
LIN {X 0,Y 409.417,Z 451.789,A -85,B 0,C 180,E1 19501.402,E2 19501.402} C_VEL
LIN {X 0,Y 409.402,Z 451.788,A -85,B 0,C 180,E1 19497.5,E2 19497.5} C_VEL
LIN {X 0,Y 409.389,Z 451.789,A -85,B 0,C 180,E1 19493.595,E2 19493.595} C_VEL
LIN {X 0,Y 409.374,Z 451.803,A -85,B 0,C 180,E1 19489.849,E2 19489.849} C_VEL
LIN {X 0,Y 409.372,Z 451.797,A -85,B 0,C 180,E1 19486.08,E2 19486.08} C_VEL
LIN {X 0,Y 409.375,Z 451.786,A -85,B 0,C 180,E1 19482.196,E2 19482.196} C_VEL
LIN {X 0,Y 409.391,Z 451.801,A -85,B 0,C 180,E1 19478.373,E2 19478.373} C_VEL
LIN {X 0,Y 409.404,Z 451.771,A -85,B 0,C 180,E1 19474.514,E2 19474.514} C_VEL
LIN {X 0,Y 409.435,Z 451.798,A -85,B 0,C 180,E1 19470.69,E2 19470.69} C_VEL
LIN {X 0,Y 409.425,Z 451.768,A -85,B 0,C 180,E1 19466.859,E2 19466.859} C_VEL
LIN {X 0,Y 409.417,Z 451.795,A -85,B 0,C 180,E1 19462.972,E2 19462.972} C_VEL
LIN {X 0,Y 409.396,Z 451.783,A -85,B 0,C 180,E1 19459.251,E2 19459.251} C_VEL
LIN {X 0,Y 409.392,Z 451.787,A -85,B 0,C 180,E1 19455.439,E2 19455.439} C_VEL
LIN {X 0,Y 409.395,Z 451.794,A -85,B 0,C 180,E1 19451.553,E2 19451.553} C_VEL
LIN {X 0,Y 409.401,Z 451.774,A -85,B 0,C 180,E1 19447.72,E2 19447.72} C_VEL
LIN {X 0,Y 409.421,Z 451.794,A -85,B 0,C 180,E1 19443.921,E2 19443.921} C_VEL
LIN {X 0,Y 409.436,Z 451.764,A -85,B 0,C 180,E1 19440,E2 19440} C_VEL
LIN {X 0,Y 409.439,Z 451.796,A -85,B 0,C 180,E1 19436.08,E2 19436.08} C_VEL
LIN {X 0,Y 409.445,Z 451.768,A -85,B 0,C 180,E1 19432.14,E2 19432.14} C_VEL
LIN {X 0,Y 409.441,Z 451.797,A -85,B 0,C 180,E1 19428.163,E2 19428.163} C_VEL
LIN {X 0,Y 409.439,Z 451.775,A -85,B 0,C 180,E1 19424.188,E2 19424.188} C_VEL
LIN {X 0,Y 409.432,Z 451.792,A -85,B 0,C 180,E1 19420.306,E2 19420.306} C_VEL
LIN {X 0,Y 409.427,Z 451.794,A -85,B 0,C 180,E1 19416.391,E2 19416.391} C_VEL
LIN {X 0,Y 409.421,Z 451.781,A -85,B 0,C 180,E1 19412.437,E2 19412.437} C_VEL
LIN {X 0,Y 409.42,Z 451.787,A -85,B 0,C 180,E1 19408.656,E2 19408.656} C_VEL
LIN {X 0,Y 409.423,Z 451.791,A -85,B 0,C 180,E1 19404.807,E2 19404.807} C_VEL
LIN {X 0,Y 409.433,Z 451.788,A -85,B 0,C 180,E1 19400.946,E2 19400.946} C_VEL
LIN {X 0,Y 409.437,Z 451.789,A -85,B 0,C 180,E1 19397.053,E2 19397.053} C_VEL
LIN {X 0,Y 409.439,Z 451.797,A -85,B 0,C 180,E1 19393.1,E2 19393.1} C_VEL
LIN {X 0,Y 409.48,Z 452.115,A -85,B 0,C 180,E1 19391.994,E2 19391.994} C_VEL
LIN {X 0,Y 417.105,Z 473.192,A -85,B 0,C 180,E1 19388.731,E2 19388.731} C_VEL
LIN {X 0,Y 424.616,Z 495.64,A -85,B 0,C 180,E1 19385.606,E2 19385.606} C_VEL
LIN {X 0,Y 420.204,Z 540.765,A -85,B 0,C 180,E1 19381.174,E2 19381.174} C_VEL
LIN {X 0,Y 422.773,Z 565.822,A -85,B 0,C 180,E1 19380.533,E2 19380.533} C_VEL
LIN {X 0,Y 419.964,Z 739.339,A -85,B 0,C 180,E1 19377.566,E2 19377.566} C_VEL
LIN {X 0,Y 419.062,Z 757.919,A -85,B 0,C 180,E1 19377.013,E2 19377.013} C_VEL
LIN {X 0,Y 417.879,Z 775.905,A -85,B 0,C 180,E1 19376.225,E2 19376.225} C_VEL
LIN {X 0,Y 416.453,Z 793.962,A -85,B 0,C 180,E1 19375.159,E2 19375.159} C_VEL
LIN {X 0,Y 414.962,Z 810.846,A -85,B 0,C 180,E1 19373.879,E2 19373.879} C_VEL
LIN {X 0,Y 413.483,Z 826.369,A -85,B 0,C 180,E1 19372.421,E2 19372.421} C_VEL
